LIN {X 0,Y 361.818,Z 305.412,A -85,B 0,C 180,E1 -12994.284,E2 -12994.284} C_VEL
LIN {X 0,Y 361.885,Z 305.409,A -85,B 0,C 180,E1 -12997.238,E2 -12997.238} C_VEL
LIN {X 0,Y 361.874,Z 305.407,A -85,B 0,C 180,E1 -13000.773,E2 -13000.773} C_VEL
LIN {X 0,Y 361.905,Z 305.409,A -85,B 0,C 180,E1 -13004.355,E2 -13004.355} C_VEL
LIN {X 0,Y 361.86,Z 305.417,A -85,B 0,C 180,E1 -13007.564,E2 -13007.564} C_VEL
LIN {X 0,Y 361.852,Z 305.412,A -85,B 0,C 180,E1 -13010.977,E2 -13010.977} C_VEL
LIN {X 0,Y 361.854,Z 305.412,A -85,B 0,C 180,E1 -13014.66,E2 -13014.66} C_VEL
LIN {X 0,Y 361.82,Z 305.42,A -85,B 0,C 180,E1 -13018.376,E2 -13018.376} C_VEL
LIN {X 0,Y 361.917,Z 305.621,A -85,B 0,C 180,E1 -13019.606,E2 -13019.606} C_VEL
LIN {X 0,Y 364.515,Z 316.864,A -85,B 0,C 180,E1 -13022.487,E2 -13022.487} C_VEL
LIN {X 0,Y 366.087,Z 325.864,A -85,B 0,C 180,E1 -13024.673,E2 -13024.673} C_VEL
LIN {X 0,Y 364.917,Z 338.677,A -85,B 0,C 180,E1 -13027.483,E2 -13027.483} C_VEL
LIN {X 0,Y 368.842,Z 360.352,A -85,B 0,C 180,E1 -13028.244,E2 -13028.244} C_VEL
LIN {X 0,Y 370.844,Z 375.541,A -85,B 0,C 180,E1 -13028.711,E2 -13028.711} C_VEL
LIN {X 0,Y 369.356,Z 448.545,A -85,B 0,C 180,E1 -13030.23,E2 -13030.23} C_VEL
LIN {X 0,Y 368.568,Z 462.077,A -85,B 0,C 180,E1 -13030.729,E2 -13030.729} C_VEL
LIN {X 0,Y 367.613,Z 474.38,A -85,B 0,C 180,E1 -13031.401,E2 -13031.401} C_VEL
LIN {X 0,Y 366.546,Z 486.228,A -85,B 0,C 180,E1 -13032.284,E2 -13032.284} C_VEL
LIN {X 0,Y 365.417,Z 497.657,A -85,B 0,C 180,E1 -13033.381,E2 -13033.381} C_VEL
LIN {X 0,Y 364.385,Z 507.488,A -85,B 0,C 180,E1 -13034.557,E2 -13034.557} C_VEL
LIN {X 0,Y 363.289,Z 517.316,A -85,B 0,C 180,E1 -13036.011,E2 -13036.011} C_VEL
LIN {X 0,Y 362.23,Z 526.378,A -85,B 0,C 180,E1 -13037.682,E2 -13037.682} C_VEL
LIN {X 0,Y 361.454,Z 533.695,A -85,B 0,C 180,E1 -13039.36,E2 -13039.36} C_VEL
LIN {X 0,Y 360.909,Z 539.555,A -85,B 0,C 180,E1 -13041.042,E2 -13041.042} C_VEL
LIN {X 0,Y 360.588,Z 544.181,A -85,B 0,C 180,E1 -13042.726,E2 -13042.726} C_VEL
LIN {X 0,Y 360.381,Z 547.708,A -85,B 0,C 180,E1 -13044.408,E2 -13044.408} C_VEL
LIN {X 0,Y 360.364,Z 549.477,A -85,B 0,C 180,E1 -13045.53,E2 -13045.53} C_VEL
LIN {X 0,Y 360.298,Z 551.789,A -85,B 0,C 180,E1 -13047.768,E2 -13047.768} C_VEL
LIN {X 0,Y 360.369,Z 552.341,A -85,B 0,C 180,E1 -13048.886,E2 -13048.886} C_VEL
LIN {X 0,Y 360.424,Z 552.454,A -85,B 0,C 180,E1 -13050.004,E2 -13050.004} C_VEL
LIN {X 0,Y 360.386,Z 552.17,A -85,B 0,C 180,E1 -13051.121,E2 -13051.121} C_VEL
LIN {X 0,Y 360.303,Z 551.492,A -85,B 0,C 180,E1 -13052.239,E2 -13052.239} C_VEL
LIN {X 0,Y 360.305,Z 550.405,A -85,B 0,C 180,E1 -13053.358,E2 -13053.358} C_VEL
LIN {X 0,Y 360.367,Z 548.86,A -85,B 0,C 180,E1 -13054.477,E2 -13054.477} C_VEL
LIN {X 0,Y 360.38,Z 546.171,A -85,B 0,C 180,E1 -13055.964,E2 -13055.964} C_VEL
LIN {X 0,Y 360.652,Z 541.532,A -85,B 0,C 180,E1 -13057.843,E2 -13057.843} C_VEL
LIN {X 0,Y 361.083,Z 535.11,A -85,B 0,C 180,E1 -13059.809,E2 -13059.809} C_VEL
LIN {X 0,Y 361.669,Z 528.101,A -85,B 0,C 180,E1 -13061.492,E2 -13061.492} C_VEL
LIN {X 0,Y 362.597,Z 519.308,A -85,B 0,C 180,E1 -13063.167,E2 -13063.167} C_VEL
LIN {X 0,Y 363.604,Z 509.036,A -85,B 0,C 180,E1 -13064.738,E2 -13064.738} C_VEL
LIN {X 0,Y 364.589,Z 497.831,A -85,B 0,C 180,E1 -13066.09,E2 -13066.09} C_VEL
LIN {X 0,Y 365.697,Z 486.255,A -85,B 0,C 180,E1 -13067.189,E2 -13067.189} C_VEL
LIN {X 0,Y 366.655,Z 474.067,A -85,B 0,C 180,E1 -13068.079,E2 -13068.079} C_VEL
LIN {X 0,Y 367.595,Z 460.562,A -85,B 0,C 180,E1 -13068.788,E2 -13068.788} C_VEL
LIN {X 0,Y 368.122,Z 448.077,A -85,B 0,C 180,E1 -13069.23,E2 -13069.23} C_VEL
LIN {X 0,Y 369.425,Z 373.616,A -85,B 0,C 180,E1 -13070.75,E2 -13070.75} C_VEL
LIN {X 0,Y 364.371,Z 340.015,A -85,B 0,C 180,E1 -13071.754,E2 -13071.754} C_VEL
LIN {X 0,Y 365.678,Z 325.548,A -85,B 0,C 180,E1 -13075.015,E2 -13075.015} C_VEL
LIN {X 0,Y 365.209,Z 321.353,A -85,B 0,C 180,E1 -13076.022,E2 -13076.022} C_VEL
LIN {X 0,Y 363.128,Z 310.962,A -85,B 0,C 180,E1 -13078.623,E2 -13078.623} C_VEL
LIN {X 0,Y 361.897,Z 305.409,A -85,B 0,C 180,E1 -13080.106,E2 -13080.106} C_VEL
LIN {X 0,Y 361.86,Z 305.412,A -85,B 0,C 180,E1 -13084.281,E2 -13084.281} C_VEL
LIN {X 0,Y 361.867,Z 305.405,A -85,B 0,C 180,E1 -13087.223,E2 -13087.223} C_VEL
LIN {X 0,Y 361.839,Z 305.411,A -85,B 0,C 180,E1 -13090.756,E2 -13090.756} C_VEL
LIN {X 0,Y 361.82,Z 305.418,A -85,B 0,C 180,E1 -13094.369,E2 -13094.369} C_VEL
LIN {X 0,Y 361.839,Z 305.409,A -85,B 0,C 180,E1 -13097.569,E2 -13097.569} C_VEL
LIN {X 0,Y 361.871,Z 305.407,A -85,B 0,C 180,E1 -13100.974,E2 -13100.974} C_VEL
LIN {X 0,Y 361.875,Z 305.411,A -85,B 0,C 180,E1 -13104.656,E2 -13104.656} C_VEL
LIN {X 0,Y 361.838,Z 305.412,A -85,B 0,C 180,E1 -13108.371,E2 -13108.371} C_VEL
LIN {X 0,Y 361.908,Z 305.401,A -85,B 0,C 180,E1 -13112.221,E2 -13112.221} C_VEL
LIN {X 0,Y 361.927,Z 305.403,A -85,B 0,C 180,E1 -13114.71,E2 -13114.71} C_VEL
LIN {X 0,Y 361.861,Z 305.407,A -85,B 0,C 180,E1 -13118.345,E2 -13118.345} C_VEL
LIN {X 0,Y 361.919,Z 305.399,A -85,B 0,C 180,E1 -13122.085,E2 -13122.085} C_VEL
LIN {X 0,Y 361.959,Z 305.398,A -85,B 0,C 180,E1 -13125.379,E2 -13125.379} C_VEL
LIN {X 0,Y 361.966,Z 305.395,A -85,B 0,C 180,E1 -13128.804,E2 -13128.804} C_VEL
LIN {X 0,Y 362.114,Z 305.374,A -85,B 0,C 180,E1 -13132.192,E2 -13132.192} C_VEL
LIN {X 0,Y 362.108,Z 305.375,A -85,B 0,C 180,E1 -13134.431,E2 -13134.431} C_VEL
LIN {X 0,Y 362.273,Z 305.358,A -85,B 0,C 180,E1 -13137.776,E2 -13137.776} C_VEL
LIN {X 0,Y 362.377,Z 305.343,A -85,B 0,C 180,E1 -13140,E2 -13140} C_VEL
LIN {X 0,Y 362.273,Z 305.355,A -85,B 0,C 180,E1 -13142.224,E2 -13142.224} C_VEL
LIN {X 0,Y 362.119,Z 305.374,A -85,B 0,C 180,E1 -13146.687,E2 -13146.687} C_VEL
LIN {X 0,Y 361.995,Z 305.392,A -85,B 0,C 180,E1 -13150.063,E2 -13150.063} C_VEL
LIN {X 0,Y 361.996,Z 305.395,A -85,B 0,C 180,E1 -13153.898,E2 -13153.898} C_VEL
LIN {X 0,Y 361.925,Z 305.398,A -85,B 0,C 180,E1 -13156.934,E2 -13156.934} C_VEL
LIN {X 0,Y 361.882,Z 305.405,A -85,B 0,C 180,E1 -13160.461,E2 -13160.461} C_VEL
LIN {X 0,Y 361.861,Z 305.413,A -85,B 0,C 180,E1 -13164.101,E2 -13164.101} C_VEL
LIN {X 0,Y 361.834,Z 305.412,A -85,B 0,C 180,E1 -13167.785,E2 -13167.785} C_VEL
LIN {X 0,Y 361.827,Z 305.41,A -85,B 0,C 180,E1 -13171.279,E2 -13171.279} C_VEL
LIN {X 0,Y 361.851,Z 305.414,A -85,B 0,C 180,E1 -13174.281,E2 -13174.281} C_VEL
LIN {X 0,Y 361.856,Z 305.407,A -85,B 0,C 180,E1 -13177.221,E2 -13177.221} C_VEL
LIN {X 0,Y 361.811,Z 305.416,A -85,B 0,C 180,E1 -13180.75,E2 -13180.75} C_VEL
LIN {X 0,Y 361.801,Z 305.418,A -85,B 0,C 180,E1 -13184.371,E2 -13184.371} C_VEL
LIN {X 0,Y 361.814,Z 305.412,A -85,B 0,C 180,E1 -13187.572,E2 -13187.572} C_VEL
LIN {X 0,Y 361.824,Z 305.414,A -85,B 0,C 180,E1 -13190.983,E2 -13190.983} C_VEL
LIN {X 0,Y 361.841,Z 305.414,A -85,B 0,C 180,E1 -13194.663,E2 -13194.663} C_VEL
LIN {X 0,Y 361.816,Z 305.413,A -85,B 0,C 180,E1 -13198.367,E2 -13198.367} C_VEL
LIN {X 0,Y 361.855,Z 305.414,A -85,B 0,C 180,E1 -13200.949,E2 -13200.949} C_VEL
LIN {X 0,Y 361.884,Z 305.406,A -85,B 0,C 180,E1 -13204.705,E2 -13204.705} C_VEL
LIN {X 0,Y 361.86,Z 305.406,A -85,B 0,C 180,E1 -13208.343,E2 -13208.343} C_VEL
LIN {X 0,Y 361.927,Z 305.398,A -85,B 0,C 180,E1 -13212.083,E2 -13212.083} C_VEL
LIN {X 0,Y 361.967,Z 305.399,A -85,B 0,C 180,E1 -13215.377,E2 -13215.377} C_VEL
LIN {X 0,Y 361.973,Z 305.393,A -85,B 0,C 180,E1 -13218.802,E2 -13218.802} C_VEL
LIN {X 0,Y 362.082,Z 305.379,A -85,B 0,C 180,E1 -13222.188,E2 -13222.188} C_VEL
LIN {X 0,Y 362.092,Z 305.377,A -85,B 0,C 180,E1 -13224.428,E2 -13224.428} C_VEL
LIN {X 0,Y 362.266,Z 305.36,A -85,B 0,C 180,E1 -13227.773,E2 -13227.773} C_VEL
LIN {X 0,Y 362.176,Z 305.368,A -85,B 0,C 180,E1 -13231.108,E2 -13231.108} C_VEL
LIN {X 0,Y 362.267,Z 305.357,A -85,B 0,C 180,E1 -13232.22,E2 -13232.22} C_VEL
LIN {X 0,Y 362.114,Z 305.379,A -85,B 0,C 180,E1 -13236.683,E2 -13236.683} C_VEL
LIN {X 0,Y 362.084,Z 305.457,A -85,B 0,C 180,E1 -13237.735,E2 -13237.735} C_VEL
LIN {X 0,Y 363.779,Z 314.594,A -85,B 0,C 180,E1 -13240.271,E2 -13240.271} C_VEL
LIN {X 0,Y 366.864,Z 324.402,A -85,B 0,C 180,E1 -13240.675,E2 -13240.675} C_VEL
LIN {X 0,Y 369.922,Z 340.115,A -85,B 0,C 180,E1 -13241.181,E2 -13241.181} C_VEL
LIN {X 0,Y 368.349,Z 422.054,A -85,B 0,C 180,E1 -13242.85,E2 -13242.85} C_VEL
LIN {X 0,Y 367.824,Z 435.697,A -85,B 0,C 180,E1 -13243.356,E2 -13243.356} C_VEL
LIN {X 0,Y 367.154,Z 448.332,A -85,B 0,C 180,E1 -13244.051,E2 -13244.051} C_VEL
LIN {X 0,Y 366.4,Z 459.282,A -85,B 0,C 180,E1 -13244.861,E2 -13244.861} C_VEL
LIN {X 0,Y 365.344,Z 471.437,A -85,B 0,C 180,E1 -13246.019,E2 -13246.019} C_VEL
LIN {X 0,Y 364.346,Z 481.673,A -85,B 0,C 180,E1 -13247.247,E2 -13247.247} C_VEL
LIN {X 0,Y 363.485,Z 491.125,A -85,B 0,C 180,E1 -13248.662,E2 -13248.662} C_VEL
LIN {X 0,Y 362.672,Z 499.049,A -85,B 0,C 180,E1 -13250.113,E2 -13250.113} C_VEL
LIN {X 0,Y 361.84,Z 507.132,A -85,B 0,C 180,E1 -13251.95,E2 -13251.95} C_VEL
LIN {X 0,Y 361.399,Z 512.236,A -85,B 0,C 180,E1 -13253.409,E2 -13253.409} C_VEL
LIN {X 0,Y 360.46,Z 514.812,A -85,B 0,C 180,E1 -13254.246,E2 -13254.246} C_VEL
LIN {X 0,Y 357.241,Z 518.482,A -85,B 0,C 180,E1 -13255.627,E2 -13255.627} C_VEL
LIN {X 0,Y 354.605,Z 520.942,A -85,B 0,C 180,E1 -13256.772,E2 -13256.772} C_VEL
LIN {X 0,Y 353.342,Z 522.719,A -85,B 0,C 180,E1 -13257.835,E2 -13257.835} C_VEL
LIN {X 0,Y 353.298,Z 522.853,A -85,B 0,C 180,E1 -13257.99,E2 -13257.99} C_VEL
LIN {X 0,Y 353.135,Z 524.909,A -85,B 0,C 180,E1 -13259.831,E2 -13259.831} C_VEL
LIN {X 0,Y 353.076,Z 525.685,A -85,B 0,C 180,E1 -13261.16,E2 -13261.16} C_VEL
LIN {X 0,Y 353.079,Z 525.823,A -85,B 0,C 180,E1 -13263.279,E2 -13263.279} C_VEL
LIN {X 0,Y 353.265,Z 524.589,A -85,B 0,C 180,E1 -13265.346,E2 -13265.346} C_VEL
LIN {X 0,Y 353.584,Z 522.143,A -85,B 0,C 180,E1 -13267.339,E2 -13267.339} C_VEL
LIN {X 0,Y 354.059,Z 518.189,A -85,B 0,C 180,E1 -13269.426,E2 -13269.426} C_VEL
LIN {X 0,Y 354.54,Z 513.776,A -85,B 0,C 180,E1 -13271.125,E2 -13271.125} C_VEL
LIN {X 0,Y 355.306,Z 507.655,A -85,B 0,C 180,E1 -13272.957,E2 -13272.957} C_VEL
LIN {X 0,Y 356.28,Z 500.017,A -85,B 0,C 180,E1 -13274.754,E2 -13274.754} C_VEL
LIN {X 0,Y 357.319,Z 492.288,A -85,B 0,C 180,E1 -13276.22,E2 -13276.22} C_VEL
LIN {X 0,Y 358.533,Z 482.581,A -85,B 0,C 180,E1 -13277.72,E2 -13277.72} C_VEL
LIN {X 0,Y 359.62,Z 471.967,A -85,B 0,C 180,E1 -13279.03,E2 -13279.03} C_VEL
LIN {X 0,Y 360.855,Z 460.512,A -85,B 0,C 180,E1 -13280.145,E2 -13280.145} C_VEL
LIN {X 0,Y 361.828,Z 448.47,A -85,B 0,C 180,E1 -13281.052,E2 -13281.052} C_VEL
LIN {X 0,Y 362.581,Z 435.556,A -85,B 0,C 180,E1 -13281.765,E2 -13281.765} C_VEL
LIN {X 0,Y 363.169,Z 422.591,A -85,B 0,C 180,E1 -13282.243,E2 -13282.243} C_VEL
LIN {X 0,Y 364.894,Z 340.765,A -85,B 0,C 180,E1 -13283.969,E2 -13283.969} C_VEL
LIN {X 0,Y 362.053,Z 327.901,A -85,B 0,C 180,E1 -13284.47,E2 -13284.47} C_VEL
LIN {X 0,Y 356.857,Z 315.027,A -85,B 0,C 180,E1 -13285.171,E2 -13285.171} C_VEL
LIN {X 0,Y 354.77,Z 306.294,A -85,B 0,C 180,E1 -13287.539,E2 -13287.539} C_VEL
LIN {X 0,Y 354.831,Z 306.29,A -85,B 0,C 180,E1 -13290.618,E2 -13290.618} C_VEL
LIN {X 0,Y 354.858,Z 306.29,A -85,B 0,C 180,E1 -13294.169,E2 -13294.169} C_VEL
LIN {X 0,Y 354.786,Z 306.298,A -85,B 0,C 180,E1 -13297.891,E2 -13297.891} C_VEL
LIN {X 0,Y 354.879,Z 306.28,A -85,B 0,C 180,E1 -13301.89,E2 -13301.89} C_VEL
LIN {X 0,Y 354.897,Z 306.277,A -85,B 0,C 180,E1 -13305.98,E2 -13305.98} C_VEL
LIN {X 0,Y 354.91,Z 306.27,A -85,B 0,C 180,E1 -13309.734,E2 -13309.734} C_VEL
LIN {X 0,Y 355.077,Z 306.253,A -85,B 0,C 180,E1 -13313.18,E2 -13313.18} C_VEL
LIN {X 0,Y 355.198,Z 306.237,A -85,B 0,C 180,E1 -13317.732,E2 -13317.732} C_VEL
LIN {X 0,Y 355.328,Z 306.214,A -85,B 0,C 180,E1 -13320,E2 -13320} C_VEL
LIN {X 0,Y 355.199,Z 306.238,A -85,B 0,C 180,E1 -13322.268,E2 -13322.268} C_VEL
LIN {X 0,Y 355.08,Z 306.252,A -85,B 0,C 180,E1 -13326.82,E2 -13326.82} C_VEL
LIN {X 0,Y 354.936,Z 306.271,A -85,B 0,C 180,E1 -13330.265,E2 -13330.265} C_VEL
LIN {X 0,Y 354.897,Z 306.275,A -85,B 0,C 180,E1 -13334.02,E2 -13334.02} C_VEL
LIN {X 0,Y 354.88,Z 306.275,A -85,B 0,C 180,E1 -13338.111,E2 -13338.111} C_VEL
LIN {X 0,Y 354.818,Z 306.282,A -85,B 0,C 180,E1 -13342.107,E2 -13342.107} C_VEL
LIN {X 0,Y 354.859,Z 306.28,A -85,B 0,C 180,E1 -13345.831,E2 -13345.831} C_VEL
LIN {X 0,Y 354.816,Z 306.288,A -85,B 0,C 180,E1 -13349.682,E2 -13349.682} C_VEL
LIN {X 0,Y 354.771,Z 306.294,A -85,B 0,C 180,E1 -13353.706,E2 -13353.706} C_VEL
LIN {X 0,Y 354.844,Z 306.283,A -85,B 0,C 180,E1 -13357.616,E2 -13357.616} C_VEL
LIN {X 0,Y 354.825,Z 306.286,A -85,B 0,C 180,E1 -13360.816,E2 -13360.816} C_VEL
LIN {X 0,Y 354.859,Z 306.286,A -85,B 0,C 180,E1 -13364.531,E2 -13364.531} C_VEL
LIN {X 0,Y 354.814,Z 306.293,A -85,B 0,C 180,E1 -13367.674,E2 -13367.674} C_VEL
LIN {X 0,Y 354.814,Z 306.289,A -85,B 0,C 180,E1 -13370.674,E2 -13370.674} C_VEL
LIN {X 0,Y 354.801,Z 306.287,A -85,B 0,C 180,E1 -13374.306,E2 -13374.306} C_VEL
LIN {X 0,Y 354.769,Z 306.303,A -85,B 0,C 180,E1 -13377.672,E2 -13377.672} C_VEL
LIN {X 0,Y 354.861,Z 306.472,A -85,B 0,C 180,E1 -13379.15,E2 -13379.15} C_VEL
LIN {X 0,Y 357.554,Z 318.013,A -85,B 0,C 180,E1 -13382.192,E2 -13382.192} C_VEL
LIN {X 0,Y 359.229,Z 327.337,A -85,B 0,C 180,E1 -13384.512,E2 -13384.512} C_VEL
LIN {X 0,Y 358.128,Z 338.37,A -85,B 0,C 180,E1 -13386.974,E2 -13386.974} C_VEL
LIN {X 0,Y 362.315,Z 360.994,A -85,B 0,C 180,E1 -13387.808,E2 -13387.808} C_VEL
LIN {X 0,Y 364.338,Z 375.808,A -85,B 0,C 180,E1 -13388.28,E2 -13388.28} C_VEL
LIN {X 0,Y 362.759,Z 448.376,A -85,B 0,C 180,E1 -13389.818,E2 -13389.818} C_VEL
LIN {X 0,Y 361.959,Z 461.864,A -85,B 0,C 180,E1 -13390.326,E2 -13390.326} C_VEL
LIN {X 0,Y 360.906,Z 474.652,A -85,B 0,C 180,E1 -13391.042,E2 -13391.042} C_VEL
LIN {X 0,Y 359.816,Z 486.378,A -85,B 0,C 180,E1 -13391.941,E2 -13391.941} C_VEL
LIN {X 0,Y 358.623,Z 497.725,A -85,B 0,C 180,E1 -13393.057,E2 -13393.057} C_VEL
LIN {X 0,Y 357.488,Z 507.837,A -85,B 0,C 180,E1 -13394.3,E2 -13394.3} C_VEL
LIN {X 0,Y 356.363,Z 517.236,A -85,B 0,C 180,E1 -13395.733,E2 -13395.733} C_VEL
LIN {X 0,Y 355.271,Z 526.256,A -85,B 0,C 180,E1 -13397.436,E2 -13397.436} C_VEL
LIN {X 0,Y 354.419,Z 533.544,A -85,B 0,C 180,E1 -13399.146,E2 -13399.146} C_VEL
LIN {X 0,Y 353.865,Z 539.378,A -85,B 0,C 180,E1 -13400.862,E2 -13400.862} C_VEL
LIN {X 0,Y 353.51,Z 543.983,A -85,B 0,C 180,E1 -13402.58,E2 -13402.58} C_VEL
LIN {X 0,Y 353.287,Z 547.494,A -85,B 0,C 180,E1 -13404.296,E2 -13404.296} C_VEL
LIN {X 0,Y 353.277,Z 549.251,A -85,B 0,C 180,E1 -13405.44,E2 -13405.44} C_VEL
LIN {X 0,Y 353.223,Z 550.597,A -85,B 0,C 180,E1 -13406.582,E2 -13406.582} C_VEL
LIN {X 0,Y 353.203,Z 551.546,A -85,B 0,C 180,E1 -13407.723,E2 -13407.723} C_VEL
LIN {X 0,Y 353.269,Z 552.081,A -85,B 0,C 180,E1 -13408.864,E2 -13408.864} C_VEL
LIN {X 0,Y 353.329,Z 552.183,A -85,B 0,C 180,E1 -13410.004,E2 -13410.004} C_VEL
LIN {X 0,Y 353.286,Z 551.89,A -85,B 0,C 180,E1 -13411.143,E2 -13411.143} C_VEL
LIN {X 0,Y 353.208,Z 551.202,A -85,B 0,C 180,E1 -13412.284,E2 -13412.284} C_VEL
LIN {X 0,Y 353.226,Z 550.096,A -85,B 0,C 180,E1 -13413.425,E2 -13413.425} C_VEL
LIN {X 0,Y 353.279,Z 548.538,A -85,B 0,C 180,E1 -13414.568,E2 -13414.568} C_VEL
LIN {X 0,Y 353.298,Z 546.122,A -85,B 0,C 180,E1 -13415.94,E2 -13415.94} C_VEL
LIN {X 0,Y 353.509,Z 542.696,A -85,B 0,C 180,E1 -13417.428,E2 -13417.428} C_VEL
LIN {X 0,Y 353.825,Z 537.689,A -85,B 0,C 180,E1 -13419.146,E2 -13419.146} C_VEL
LIN {X 0,Y 354.334,Z 531.382,A -85,B 0,C 180,E1 -13420.864,E2 -13420.864} C_VEL
LIN {X 0,Y 355.152,Z 523.483,A -85,B 0,C 180,E1 -13422.575,E2 -13422.575} C_VEL
LIN {X 0,Y 355.985,Z 515.412,A -85,B 0,C 180,E1 -13423.998,E2 -13423.998} C_VEL
LIN {X 0,Y 356.98,Z 505.448,A -85,B 0,C 180,E1 -13425.431,E2 -13425.431} C_VEL
LIN {X 0,Y 358.019,Z 494.582,A -85,B 0,C 180,E1 -13426.687,E2 -13426.687} C_VEL
LIN {X 0,Y 359.162,Z 482.061,A -85,B 0,C 180,E1 -13427.806,E2 -13427.806} C_VEL
LIN {X 0,Y 360.153,Z 469.789,A -85,B 0,C 180,E1 -13428.638,E2 -13428.638} C_VEL
LIN {X 0,Y 360.946,Z 456.887,A -85,B 0,C 180,E1 -13429.259,E2 -13429.259} C_VEL
LIN {X 0,Y 361.503,Z 443.35,A -85,B 0,C 180,E1 -13429.671,E2 -13429.671} C_VEL
LIN {X 0,Y 362.658,Z 374.276,A -85,B 0,C 180,E1 -13431.097,E2 -13431.097} C_VEL
LIN {X 0,Y 357.485,Z 339.682,A -85,B 0,C 180,E1 -13432.174,E2 -13432.174} C_VEL
LIN {X 0,Y 358.732,Z 326.411,A -85,B 0,C 180,E1 -13435.223,E2 -13435.223} C_VEL
LIN {X 0,Y 357.763,Z 319.8,A -85,B 0,C 180,E1 -13436.862,E2 -13436.862} C_VEL
LIN {X 0,Y 354.862,Z 306.286,A -85,B 0,C 180,E1 -13440.417,E2 -13440.417} C_VEL
LIN {X 0,Y 354.812,Z 306.286,A -85,B 0,C 180,E1 -13443.703,E2 -13443.703} C_VEL
LIN {X 0,Y 354.803,Z 306.289,A -85,B 0,C 180,E1 -13446.461,E2 -13446.461} C_VEL
LIN {X 0,Y 354.83,Z 306.282,A -85,B 0,C 180,E1 -13449.424,E2 -13449.424} C_VEL
LIN {X 0,Y 354.792,Z 306.288,A -85,B 0,C 180,E1 -13452.868,E2 -13452.868} C_VEL
LIN {X 0,Y 354.77,Z 306.292,A -85,B 0,C 180,E1 -13456.104,E2 -13456.104} C_VEL
LIN {X 0,Y 354.79,Z 306.288,A -85,B 0,C 180,E1 -13459.179,E2 -13459.179} C_VEL
LIN {X 0,Y 354.809,Z 306.289,A -85,B 0,C 180,E1 -13462.403,E2 -13462.403} C_VEL
LIN {X 0,Y 354.813,Z 306.288,A -85,B 0,C 180,E1 -13464.941,E2 -13464.941} C_VEL
LIN {X 0,Y 354.794,Z 306.289,A -85,B 0,C 180,E1 -13468.406,E2 -13468.406} C_VEL
LIN {X 0,Y 354.847,Z 306.28,A -85,B 0,C 180,E1 -13471.619,E2 -13471.619} C_VEL
LIN {X 0,Y 354.898,Z 306.274,A -85,B 0,C 180,E1 -13474.172,E2 -13474.172} C_VEL
LIN {X 0,Y 354.816,Z 306.284,A -85,B 0,C 180,E1 -13477.893,E2 -13477.893} C_VEL
LIN {X 0,Y 354.889,Z 306.275,A -85,B 0,C 180,E1 -13481.908,E2 -13481.908} C_VEL
LIN {X 0,Y 354.941,Z 306.268,A -85,B 0,C 180,E1 -13485.982,E2 -13485.982} C_VEL
LIN {X 0,Y 354.954,Z 306.268,A -85,B 0,C 180,E1 -13489.735,E2 -13489.735} C_VEL
LIN {X 0,Y 355.121,Z 306.251,A -85,B 0,C 180,E1 -13493.18,E2 -13493.18} C_VEL
LIN {X 0,Y 355.237,Z 306.235,A -85,B 0,C 180,E1 -13497.732,E2 -13497.732} C_VEL
LIN {X 0,Y 355.328,Z 306.221,A -85,B 0,C 180,E1 -13500,E2 -13500} C_VEL
LIN {X 0,Y 355.237,Z 306.232,A -85,B 0,C 180,E1 -13502.268,E2 -13502.268} C_VEL
LIN {X 0,Y 355.084,Z 306.25,A -85,B 0,C 180,E1 -13506.82,E2 -13506.82} C_VEL
LIN {X 0,Y 354.952,Z 306.268,A -85,B 0,C 180,E1 -13510.265,E2 -13510.265} C_VEL
LIN {X 0,Y 354.941,Z 306.273,A -85,B 0,C 180,E1 -13514.018,E2 -13514.018} C_VEL
LIN {X 0,Y 354.889,Z 306.279,A -85,B 0,C 180,E1 -13518.092,E2 -13518.092} C_VEL
LIN {X 0,Y 354.804,Z 306.291,A -85,B 0,C 180,E1 -13522.108,E2 -13522.108} C_VEL
LIN {X 0,Y 354.794,Z 306.29,A -85,B 0,C 180,E1 -13525.836,E2 -13525.836} C_VEL
LIN {X 0,Y 354.786,Z 306.289,A -85,B 0,C 180,E1 -13529.685,E2 -13529.685} C_VEL
LIN {X 0,Y 354.809,Z 306.286,A -85,B 0,C 180,E1 -13533.702,E2 -13533.702} C_VEL
LIN {X 0,Y 354.792,Z 306.292,A -85,B 0,C 180,E1 -13536.46,E2 -13536.46} C_VEL
LIN {X 0,Y 354.771,Z 306.289,A -85,B 0,C 180,E1 -13539.412,E2 -13539.412} C_VEL
LIN {X 0,Y 354.78,Z 306.291,A -85,B 0,C 180,E1 -13542.865,E2 -13542.865} C_VEL
LIN {X 0,Y 354.741,Z 306.295,A -85,B 0,C 180,E1 -13546.098,E2 -13546.098} C_VEL
LIN {X 0,Y 354.765,Z 306.292,A -85,B 0,C 180,E1 -13549.174,E2 -13549.174} C_VEL
LIN {X 0,Y 354.787,Z 306.29,A -85,B 0,C 180,E1 -13552.407,E2 -13552.407} C_VEL
LIN {X 0,Y 354.776,Z 306.294,A -85,B 0,C 180,E1 -13554.935,E2 -13554.935} C_VEL
LIN {X 0,Y 354.772,Z 306.291,A -85,B 0,C 180,E1 -13558.411,E2 -13558.411} C_VEL
LIN {X 0,Y 354.794,Z 306.287,A -85,B 0,C 180,E1 -13561.612,E2 -13561.612} C_VEL
LIN {X 0,Y 354.84,Z 306.282,A -85,B 0,C 180,E1 -13565.656,E2 -13565.656} C_VEL
LIN {X 0,Y 354.833,Z 306.288,A -85,B 0,C 180,E1 -13569.111,E2 -13569.111} C_VEL
LIN {X 0,Y 354.886,Z 306.277,A -85,B 0,C 180,E1 -13572.717,E2 -13572.717} C_VEL
LIN {X 0,Y 354.957,Z 306.266,A -85,B 0,C 180,E1 -13576.253,E2 -13576.253} C_VEL
LIN {X 0,Y 354.958,Z 306.269,A -85,B 0,C 180,E1 -13579.732,E2 -13579.732} C_VEL
LIN {X 0,Y 355.089,Z 306.253,A -85,B 0,C 180,E1 -13583.177,E2 -13583.177} C_VEL
LIN {X 0,Y 355.229,Z 306.237,A -85,B 0,C 180,E1 -13587.729,E2 -13587.729} C_VEL
LIN {X 0,Y 355.147,Z 306.244,A -85,B 0,C 180,E1 -13591.13,E2 -13591.13} C_VEL
LIN {X 0,Y 355.229,Z 306.233,A -85,B 0,C 180,E1 -13592.264,E2 -13592.264} C_VEL
LIN {X 0,Y 355.079,Z 306.255,A -85,B 0,C 180,E1 -13596.816,E2 -13596.816} C_VEL
LIN {X 0,Y 355.038,Z 306.425,A -85,B 0,C 180,E1 -13597.46,E2 -13597.46} C_VEL
LIN {X 0,Y 356.696,Z 315.172,A -85,B 0,C 180,E1 -13599.884,E2 -13599.884} C_VEL
LIN {X 0,Y 360.429,Z 326.619,A -85,B 0,C 180,E1 -13600.355,E2 -13600.355} C_VEL
LIN {X 0,Y 363.224,Z 341.58,A -85,B 0,C 180,E1 -13600.841,E2 -13600.841} C_VEL
LIN {X 0,Y 361.555,Z 422.92,A -85,B 0,C 180,E1 -13602.535,E2 -13602.535} C_VEL
LIN {X 0,Y 361.012,Z 436.623,A -85,B 0,C 180,E1 -13603.063,E2 -13603.063} C_VEL
LIN {X 0,Y 360.333,Z 448.699,A -85,B 0,C 180,E1 -13603.747,E2 -13603.747} C_VEL
LIN {X 0,Y 359.556,Z 459.617,A -85,B 0,C 180,E1 -13604.571,E2 -13604.571} C_VEL
LIN {X 0,Y 358.556,Z 470.653,A -85,B 0,C 180,E1 -13605.63,E2 -13605.63} C_VEL
LIN {X 0,Y 357.465,Z 481.855,A -85,B 0,C 180,E1 -13606.985,E2 -13606.985} C_VEL
LIN {X 0,Y 356.6,Z 491.031,A -85,B 0,C 180,E1 -13608.376,E2 -13608.376} C_VEL
LIN {X 0,Y 355.685,Z 499.347,A -85,B 0,C 180,E1 -13609.923,E2 -13609.923} C_VEL
LIN {X 0,Y 354.839,Z 507.208,A -85,B 0,C 180,E1 -13611.74,E2 -13611.74} C_VEL
LIN {X 0,Y 354.344,Z 512.793,A -85,B 0,C 180,E1 -13613.365,E2 -13613.365} C_VEL
LIN {X 0,Y 353.843,Z 517.933,A -85,B 0,C 180,E1 -13615.273,E2 -13615.273} C_VEL
LIN {X 0,Y 353.442,Z 521.739,A -85,B 0,C 180,E1 -13617.21,E2 -13617.21} C_VEL
LIN {X 0,Y 353.298,Z 522.853,A -85,B 0,C 180,E1 -13617.99,E2 -13617.99} C_VEL
LIN {X 0,Y 352.513,Z 524.096,A -85,B 0,C 180,E1 -13618.92,E2 -13618.92} C_VEL
LIN {X 0,Y 349.512,Z 525.486,A -85,B 0,C 180,E1 -13620.446,E2 -13620.446} C_VEL
LIN {X 0,Y 347.056,Z 526.065,A -85,B 0,C 180,E1 -13621.692,E2 -13621.692} C_VEL
LIN {X 0,Y 346.046,Z 526.177,A -85,B 0,C 180,E1 -13622.66,E2 -13622.66} C_VEL
LIN {X 0,Y 345.985,Z 526.114,A -85,B 0,C 180,E1 -13622.988,E2 -13622.988} C_VEL
LIN {X 0,Y 346.093,Z 525.472,A -85,B 0,C 180,E1 -13624.644,E2 -13624.644} C_VEL
LIN {X 0,Y 346.278,Z 524.291,A -85,B 0,C 180,E1 -13626.049,E2 -13626.049} C_VEL
LIN {X 0,Y 346.673,Z 521.119,A -85,B 0,C 180,E1 -13628.276,E2 -13628.276} C_VEL
LIN {X 0,Y 347.242,Z 516.699,A -85,B 0,C 180,E1 -13630.357,E2 -13630.357} C_VEL
LIN {X 0,Y 347.898,Z 511.49,A -85,B 0,C 180,E1 -13632.189,E2 -13632.189} C_VEL
LIN {X 0,Y 348.822,Z 504.634,A -85,B 0,C 180,E1 -13634.06,E2 -13634.06} C_VEL
LIN {X 0,Y 349.875,Z 497.053,A -85,B 0,C 180,E1 -13635.71,E2 -13635.71} C_VEL
LIN {X 0,Y 351.132,Z 487.729,A -85,B 0,C 180,E1 -13637.347,E2 -13637.347} C_VEL
LIN {X 0,Y 352.296,Z 477.92,A -85,B 0,C 180,E1 -13638.728,E2 -13638.728} C_VEL
LIN {X 0,Y 353.529,Z 467.246,A -85,B 0,C 180,E1 -13639.929,E2 -13639.929} C_VEL
LIN {X 0,Y 354.579,Z 455.84,A -85,B 0,C 180,E1 -13640.951,E2 -13640.951} C_VEL
LIN {X 0,Y 355.583,Z 443.757,A -85,B 0,C 180,E1 -13641.77,E2 -13641.77} C_VEL
LIN {X 0,Y 356.217,Z 430.494,A -85,B 0,C 180,E1 -13642.417,E2 -13642.417} C_VEL
LIN {X 0,Y 356.801,Z 417.101,A -85,B 0,C 180,E1 -13642.815,E2 -13642.815} C_VEL
LIN {X 0,Y 358.493,Z 342.127,A -85,B 0,C 180,E1 -13644.408,E2 -13644.408} C_VEL
LIN {X 0,Y 355.846,Z 330.29,A -85,B 0,C 180,E1 -13644.885,E2 -13644.885} C_VEL
LIN {X 0,Y 349.7,Z 315.268,A -85,B 0,C 180,E1 -13645.756,E2 -13645.756} C_VEL
LIN {X 0,Y 347.715,Z 307.175,A -85,B 0,C 180,E1 -13648.044,E2 -13648.044} C_VEL
LIN {X 0,Y 347.767,Z 307.168,A -85,B 0,C 180,E1 -13650.986,E2 -13650.986} C_VEL
LIN {X 0,Y 347.791,Z 307.169,A -85,B 0,C 180,E1 -13653.604,E2 -13653.604} C_VEL
LIN {X 0,Y 347.746,Z 307.176,A -85,B 0,C 180,E1 -13656.159,E2 -13656.159} C_VEL
LIN {X 0,Y 347.761,Z 307.17,A -85,B 0,C 180,E1 -13659.906,E2 -13659.906} C_VEL
LIN {X 0,Y 347.822,Z 307.162,A -85,B 0,C 180,E1 -13662.357,E2 -13662.357} C_VEL
LIN {X 0,Y 347.853,Z 307.155,A -85,B 0,C 180,E1 -13665.969,E2 -13665.969} C_VEL
LIN {X 0,Y 347.85,Z 307.15,A -85,B 0,C 180,E1 -13669.523,E2 -13669.523} C_VEL
LIN {X 0,Y 348.043,Z 307.128,A -85,B 0,C 180,E1 -13673.041,E2 -13673.041} C_VEL
LIN {X 0,Y 348.161,Z 307.114,A -85,B 0,C 180,E1 -13677.686,E2 -13677.686} C_VEL
LIN {X 0,Y 348.278,Z 307.092,A -85,B 0,C 180,E1 -13680,E2 -13680} C_VEL
LIN {X 0,Y 348.161,Z 307.115,A -85,B 0,C 180,E1 -13682.314,E2 -13682.314} C_VEL
LIN {X 0,Y 348.046,Z 307.126,A -85,B 0,C 180,E1 -13686.959,E2 -13686.959} C_VEL
LIN {X 0,Y 347.887,Z 307.15,A -85,B 0,C 180,E1 -13690.476,E2 -13690.476} C_VEL
LIN {X 0,Y 347.854,Z 307.152,A -85,B 0,C 180,E1 -13694.152,E2 -13694.152} C_VEL
LIN {X 0,Y 347.849,Z 307.151,A -85,B 0,C 180,E1 -13698.293,E2 -13698.293} C_VEL
LIN {X 0,Y 347.781,Z 307.161,A -85,B 0,C 180,E1 -13701.652,E2 -13701.652} C_VEL
LIN {X 0,Y 347.78,Z 307.155,A -85,B 0,C 180,E1 -13705.111,E2 -13705.111} C_VEL
LIN {X 0,Y 347.772,Z 307.157,A -85,B 0,C 180,E1 -13707.697,E2 -13707.697} C_VEL
LIN {X 0,Y 347.726,Z 307.168,A -85,B 0,C 180,E1 -13710.35,E2 -13710.35} C_VEL
LIN {X 0,Y 347.711,Z 307.169,A -85,B 0,C 180,E1 -13714.468,E2 -13714.468} C_VEL
LIN {X 0,Y 347.804,Z 307.158,A -85,B 0,C 180,E1 -13718.006,E2 -13718.006} C_VEL
LIN {X 0,Y 347.754,Z 307.17,A -85,B 0,C 180,E1 -13721.83,E2 -13721.83} C_VEL
LIN {X 0,Y 347.803,Z 307.166,A -85,B 0,C 180,E1 -13725.011,E2 -13725.011} C_VEL
LIN {X 0,Y 347.759,Z 307.169,A -85,B 0,C 180,E1 -13728.396,E2 -13728.396} C_VEL
LIN {X 0,Y 347.754,Z 307.168,A -85,B 0,C 180,E1 -13732.016,E2 -13732.016} C_VEL
LIN {X 0,Y 347.725,Z 307.176,A -85,B 0,C 180,E1 -13735.541,E2 -13735.541} C_VEL
LIN {X 0,Y 347.754,Z 307.246,A -85,B 0,C 180,E1 -13738.648,E2 -13738.648} C_VEL
LIN {X 0,Y 350.485,Z 318.512,A -85,B 0,C 180,E1 -13741.707,E2 -13741.707} C_VEL
LIN {X 0,Y 352.347,Z 328.625,A -85,B 0,C 180,E1 -13744.295,E2 -13744.295} C_VEL
LIN {X 0,Y 351.388,Z 338.051,A -85,B 0,C 180,E1 -13746.446,E2 -13746.446} C_VEL
LIN {X 0,Y 355.865,Z 362.01,A -85,B 0,C 180,E1 -13747.359,E2 -13747.359} C_VEL
LIN {X 0,Y 357.847,Z 376.7,A -85,B 0,C 180,E1 -13747.844,E2 -13747.844} C_VEL
LIN {X 0,Y 356.199,Z 447.1,A -85,B 0,C 180,E1 -13749.354,E2 -13749.354} C_VEL
LIN {X 0,Y 355.441,Z 460.897,A -85,B 0,C 180,E1 -13749.874,E2 -13749.874} C_VEL
LIN {X 0,Y 354.334,Z 473.91,A -85,B 0,C 180,E1 -13750.601,E2 -13750.601} C_VEL
LIN {X 0,Y 353.093,Z 486.528,A -85,B 0,C 180,E1 -13751.585,E2 -13751.585} C_VEL
LIN {X 0,Y 351.843,Z 497.8,A -85,B 0,C 180,E1 -13752.72,E2 -13752.72} C_VEL
LIN {X 0,Y 350.661,Z 507.6,A -85,B 0,C 180,E1 -13753.951,E2 -13753.951} C_VEL
LIN {X 0,Y 349.445,Z 517.185,A -85,B 0,C 180,E1 -13755.445,E2 -13755.445} C_VEL
LIN {X 0,Y 348.321,Z 526.171,A -85,B 0,C 180,E1 -13757.181,E2 -13757.181} C_VEL
LIN {X 0,Y 347.411,Z 533.416,A -85,B 0,C 180,E1 -13758.924,E2 -13758.924} C_VEL
LIN {X 0,Y 346.836,Z 539.21,A -85,B 0,C 180,E1 -13760.675,E2 -13760.675} C_VEL
LIN {X 0,Y 346.46,Z 543.787,A -85,B 0,C 180,E1 -13762.428,E2 -13762.428} C_VEL
LIN {X 0,Y 346.198,Z 547.278,A -85,B 0,C 180,E1 -13764.179,E2 -13764.179} C_VEL
LIN {X 0,Y 346.173,Z 549.025,A -85,B 0,C 180,E1 -13765.346,E2 -13765.346} C_VEL
LIN {X 0,Y 346.147,Z 550.364,A -85,B 0,C 180,E1 -13766.512,E2 -13766.512} C_VEL
LIN {X 0,Y 346.112,Z 551.304,A -85,B 0,C 180,E1 -13767.676,E2 -13767.676} C_VEL
LIN {X 0,Y 346.17,Z 551.819,A -85,B 0,C 180,E1 -13768.841,E2 -13768.841} C_VEL
LIN {X 0,Y 346.234,Z 551.913,A -85,B 0,C 180,E1 -13770.004,E2 -13770.004} C_VEL
LIN {X 0,Y 346.187,Z 551.61,A -85,B 0,C 180,E1 -13771.167,E2 -13771.167} C_VEL
LIN {X 0,Y 346.117,Z 550.912,A -85,B 0,C 180,E1 -13772.331,E2 -13772.331} C_VEL
LIN {X 0,Y 346.15,Z 549.786,A -85,B 0,C 180,E1 -13773.496,E2 -13773.496} C_VEL
LIN {X 0,Y 346.194,Z 548.216,A -85,B 0,C 180,E1 -13774.661,E2 -13774.661} C_VEL
LIN {X 0,Y 346.247,Z 545.044,A -85,B 0,C 180,E1 -13776.412,E2 -13776.412} C_VEL
LIN {X 0,Y 346.522,Z 540.789,A -85,B 0,C 180,E1 -13778.165,E2 -13778.165} C_VEL
LIN {X 0,Y 347.027,Z 534.31,A -85,B 0,C 180,E1 -13780.21,E2 -13780.21} C_VEL
LIN {X 0,Y 347.699,Z 527.214,A -85,B 0,C 180,E1 -13781.96,E2 -13781.96} C_VEL
LIN {X 0,Y 348.649,Z 518.327,A -85,B 0,C 180,E1 -13783.704,E2 -13783.704} C_VEL
LIN {X 0,Y 349.655,Z 509.221,A -85,B 0,C 180,E1 -13785.15,E2 -13785.15} C_VEL
LIN {X 0,Y 350.614,Z 499.174,A -85,B 0,C 180,E1 -13786.45,E2 -13786.45} C_VEL
LIN {X 0,Y 351.773,Z 488.02,A -85,B 0,C 180,E1 -13787.591,E2 -13787.591} C_VEL
LIN {X 0,Y 352.877,Z 475.532,A -85,B 0,C 180,E1 -13788.585,E2 -13788.585} C_VEL
LIN {X 0,Y 353.819,Z 462.882,A -85,B 0,C 180,E1 -13789.323,E2 -13789.323} C_VEL
LIN {X 0,Y 354.519,Z 449.556,A -85,B 0,C 180,E1 -13789.848,E2 -13789.848} C_VEL
LIN {X 0,Y 355.319,Z 417.401,A -85,B 0,C 180,E1 -13790.556,E2 -13790.556} C_VEL
LIN {X 0,Y 355.915,Z 374.589,A -85,B 0,C 180,E1 -13791.465,E2 -13791.465} C_VEL
LIN {X 0,Y 350.626,Z 339.534,A -85,B 0,C 180,E1 -13792.559,E2 -13792.559} C_VEL
LIN {X 0,Y 351.797,Z 327.391,A -85,B 0,C 180,E1 -13795.409,E2 -13795.409} C_VEL
LIN {X 0,Y 350.421,Z 319.314,A -85,B 0,C 180,E1 -13797.472,E2 -13797.472} C_VEL
LIN {X 0,Y 347.79,Z 307.164,A -85,B 0,C 180,E1 -13800.724,E2 -13800.724} C_VEL
LIN {X 0,Y 347.75,Z 307.167,A -85,B 0,C 180,E1 -13804.465,E2 -13804.465} C_VEL
LIN {X 0,Y 347.777,Z 307.164,A -85,B 0,C 180,E1 -13807.989,E2 -13807.989} C_VEL
LIN {X 0,Y 347.755,Z 307.165,A -85,B 0,C 180,E1 -13811.831,E2 -13811.831} C_VEL
LIN {X 0,Y 347.708,Z 307.17,A -85,B 0,C 180,E1 -13815.028,E2 -13815.028} C_VEL
LIN {X 0,Y 347.753,Z 307.169,A -85,B 0,C 180,E1 -13818.398,E2 -13818.398} C_VEL
LIN {X 0,Y 347.776,Z 307.162,A -85,B 0,C 180,E1 -13822.012,E2 -13822.012} C_VEL
LIN {X 0,Y 347.746,Z 307.164,A -85,B 0,C 180,E1 -13825.536,E2 -13825.536} C_VEL
LIN {X 0,Y 347.746,Z 307.167,A -85,B 0,C 180,E1 -13828.3,E2 -13828.3} C_VEL
LIN {X 0,Y 347.779,Z 307.165,A -85,B 0,C 180,E1 -13830.988,E2 -13830.988} C_VEL
LIN {X 0,Y 347.83,Z 307.154,A -85,B 0,C 180,E1 -13833.608,E2 -13833.608} C_VEL
LIN {X 0,Y 347.786,Z 307.16,A -85,B 0,C 180,E1 -13836.162,E2 -13836.162} C_VEL
LIN {X 0,Y 347.784,Z 307.16,A -85,B 0,C 180,E1 -13839.908,E2 -13839.908} C_VEL
LIN {X 0,Y 347.829,Z 307.156,A -85,B 0,C 180,E1 -13843.568,E2 -13843.568} C_VEL
LIN {X 0,Y 347.886,Z 307.153,A -85,B 0,C 180,E1 -13847.16,E2 -13847.16} C_VEL
LIN {X 0,Y 348.042,Z 307.13,A -85,B 0,C 180,E1 -13851.67,E2 -13851.67} C_VEL
LIN {X 0,Y 348.057,Z 307.126,A -85,B 0,C 180,E1 -13854.206,E2 -13854.206} C_VEL
LIN {X 0,Y 348.199,Z 307.112,A -85,B 0,C 180,E1 -13857.686,E2 -13857.686} C_VEL
LIN {X 0,Y 348.28,Z 307.099,A -85,B 0,C 180,E1 -13860,E2 -13860} C_VEL
LIN {X 0,Y 348.199,Z 307.108,A -85,B 0,C 180,E1 -13862.314,E2 -13862.314} C_VEL
LIN {X 0,Y 348.051,Z 307.127,A -85,B 0,C 180,E1 -13866.959,E2 -13866.959} C_VEL
LIN {X 0,Y 347.892,Z 307.147,A -85,B 0,C 180,E1 -13870.476,E2 -13870.476} C_VEL
LIN {X 0,Y 347.899,Z 307.148,A -85,B 0,C 180,E1 -13874.15,E2 -13874.15} C_VEL
LIN {X 0,Y 347.828,Z 307.157,A -85,B 0,C 180,E1 -13878.259,E2 -13878.259} C_VEL
LIN {X 0,Y 347.762,Z 307.165,A -85,B 0,C 180,E1 -13881.624,E2 -13881.624} C_VEL
LIN {X 0,Y 347.732,Z 307.166,A -85,B 0,C 180,E1 -13885.115,E2 -13885.115} C_VEL
LIN {X 0,Y 347.724,Z 307.169,A -85,B 0,C 180,E1 -13887.701,E2 -13887.701} C_VEL
LIN {X 0,Y 347.727,Z 307.172,A -85,B 0,C 180,E1 -13890.35,E2 -13890.35} C_VEL
LIN {X 0,Y 347.75,Z 307.168,A -85,B 0,C 180,E1 -13894.043,E2 -13894.043} C_VEL
LIN {X 0,Y 347.755,Z 307.163,A -85,B 0,C 180,E1 -13897.322,E2 -13897.322} C_VEL
LIN {X 0,Y 347.698,Z 307.175,A -85,B 0,C 180,E1 -13900.302,E2 -13900.302} C_VEL
LIN {X 0,Y 347.72,Z 307.168,A -85,B 0,C 180,E1 -13903.409,E2 -13903.409} C_VEL
LIN {X 0,Y 347.715,Z 307.174,A -85,B 0,C 180,E1 -13906.688,E2 -13906.688} C_VEL
LIN {X 0,Y 347.705,Z 307.171,A -85,B 0,C 180,E1 -13910.182,E2 -13910.182} C_VEL
LIN {X 0,Y 347.742,Z 307.171,A -85,B 0,C 180,E1 -13912.675,E2 -13912.675} C_VEL
LIN {X 0,Y 347.73,Z 307.166,A -85,B 0,C 180,E1 -13915.961,E2 -13915.961} C_VEL
LIN {X 0,Y 347.733,Z 307.166,A -85,B 0,C 180,E1 -13919.649,E2 -13919.649} C_VEL
LIN {X 0,Y 347.743,Z 307.166,A -85,B 0,C 180,E1 -13923.598,E2 -13923.598} C_VEL
LIN {X 0,Y 347.768,Z 307.162,A -85,B 0,C 180,E1 -13926.158,E2 -13926.158} C_VEL
LIN {X 0,Y 347.806,Z 307.157,A -85,B 0,C 180,E1 -13929.906,E2 -13929.906} C_VEL
LIN {X 0,Y 347.837,Z 307.156,A -85,B 0,C 180,E1 -13933.566,E2 -13933.566} C_VEL
LIN {X 0,Y 347.895,Z 307.151,A -85,B 0,C 180,E1 -13937.158,E2 -13937.158} C_VEL
LIN {X 0,Y 347.939,Z 307.141,A -85,B 0,C 180,E1 -13940.698,E2 -13940.698} C_VEL
LIN {X 0,Y 348.04,Z 307.128,A -85,B 0,C 180,E1 -13944.202,E2 -13944.202} C_VEL
LIN {X 0,Y 348.19,Z 307.114,A -85,B 0,C 180,E1 -13947.683,E2 -13947.683} C_VEL
LIN {X 0,Y 348.118,Z 307.12,A -85,B 0,C 180,E1 -13951.153,E2 -13951.153} C_VEL
LIN {X 0,Y 348.191,Z 307.11,A -85,B 0,C 180,E1 -13952.31,E2 -13952.31} C_VEL
LIN {X 0,Y 348.045,Z 307.131,A -85,B 0,C 180,E1 -13956.955,E2 -13956.955} C_VEL
LIN {X 0,Y 348.036,Z 307.332,A -85,B 0,C 180,E1 -13957.173,E2 -13957.173} C_VEL
LIN {X 0,Y 349.515,Z 315.17,A -85,B 0,C 180,E1 -13959.435,E2 -13959.435} C_VEL
LIN {X 0,Y 353.87,Z 328.161,A -85,B 0,C 180,E1 -13960.003,E2 -13960.003} C_VEL
LIN {X 0,Y 356.533,Z 342.065,A -85,B 0,C 180,E1 -13960.47,E2 -13960.47} C_VEL
LIN {X 0,Y 354.812,Z 422.814,A -85,B 0,C 180,E1 -13962.181,E2 -13962.181} C_VEL
LIN {X 0,Y 354.234,Z 436.896,A -85,B 0,C 180,E1 -13962.73,E2 -13962.73} C_VEL
LIN {X 0,Y 353.527,Z 449.202,A -85,B 0,C 180,E1 -13963.443,E2 -13963.443} C_VEL
LIN {X 0,Y 352.56,Z 461.652,A -85,B 0,C 180,E1 -13964.424,E2 -13964.424} C_VEL
LIN {X 0,Y 351.497,Z 473.471,A -85,B 0,C 180,E1 -13965.629,E2 -13965.629} C_VEL
LIN {X 0,Y 350.308,Z 484.431,A -85,B 0,C 180,E1 -13967.057,E2 -13967.057} C_VEL
LIN {X 0,Y 349.413,Z 493.135,A -85,B 0,C 180,E1 -13968.464,E2 -13968.464} C_VEL
LIN {X 0,Y 348.57,Z 501.122,A -85,B 0,C 180,E1 -13970.04,E2 -13970.04} C_VEL
LIN {X 0,Y 347.8,Z 507.736,A -85,B 0,C 180,E1 -13971.639,E2 -13971.639} C_VEL
LIN {X 0,Y 347.294,Z 513.086,A -85,B 0,C 180,E1 -13973.236,E2 -13973.236} C_VEL
LIN {X 0,Y 346.797,Z 518.212,A -85,B 0,C 180,E1 -13975.181,E2 -13975.181} C_VEL
LIN {X 0,Y 346.435,Z 521.44,A -85,B 0,C 180,E1 -13976.796,E2 -13976.796} C_VEL
LIN {X 0,Y 346.21,Z 523.18,A -85,B 0,C 180,E1 -13977.949,E2 -13977.949} C_VEL
LIN {X 0,Y 346.093,Z 524.596,A -85,B 0,C 180,E1 -13979.168,E2 -13979.168} C_VEL
LIN {X 0,Y 345.962,Z 526.058,A -85,B 0,C 180,E1 -13981.438,E2 -13981.438} C_VEL
LIN {X 0,Y 345.985,Z 526.114,A -85,B 0,C 180,E1 -13982.988,E2 -13982.988} C_VEL
LIN {X 0,Y 345.388,Z 525.928,A -85,B 0,C 180,E1 -13983.96,E2 -13983.96} C_VEL
LIN {X 0,Y 342.657,Z 524.965,A -85,B 0,C 180,E1 -13985.539,E2 -13985.539} C_VEL
LIN {X 0,Y 340.401,Z 523.751,A -85,B 0,C 180,E1 -13986.808,E2 -13986.808} C_VEL
LIN {X 0,Y 339.552,Z 522.479,A -85,B 0,C 180,E1 -13987.778,E2 -13987.778} C_VEL
LIN {X 0,Y 339.549,Z 521.985,A -85,B 0,C 180,E1 -13988.104,E2 -13988.104} C_VEL
LIN {X 0,Y 340.081,Z 518.031,A -85,B 0,C 180,E1 -13990.126,E2 -13990.126} C_VEL
LIN {X 0,Y 340.8,Z 512.898,A -85,B 0,C 180,E1 -13992.064,E2 -13992.064} C_VEL
LIN {X 0,Y 341.691,Z 506.461,A -85,B 0,C 180,E1 -13993.954,E2 -13993.954} C_VEL
LIN {X 0,Y 342.89,Z 498.333,A -85,B 0,C 180,E1 -13995.828,E2 -13995.828} C_VEL
LIN {X 0,Y 344.028,Z 490.206,A -85,B 0,C 180,E1 -13997.333,E2 -13997.333} C_VEL
LIN {X 0,Y 345.363,Z 480.228,A -85,B 0,C 180,E1 -13998.835,E2 -13998.835} C_VEL
LIN {X 0,Y 346.603,Z 469.941,A -85,B 0,C 180,E1 -14000.08,E2 -14000.08} C_VEL
LIN {X 0,Y 347.807,Z 458.009,A -85,B 0,C 180,E1 -14001.214,E2 -14001.214} C_VEL
LIN {X 0,Y 348.91,Z 445.594,A -85,B 0,C 180,E1 -14002.111,E2 -14002.111} C_VEL
LIN {X 0,Y 349.627,Z 433.5,A -85,B 0,C 180,E1 -14002.751,E2 -14002.751} C_VEL
LIN {X 0,Y 350.214,Z 419.935,A -85,B 0,C 180,E1 -14003.207,E2 -14003.207} C_VEL
LIN {X 0,Y 352.027,Z 342.989,A -85,B 0,C 180,E1 -14004.883,E2 -14004.883} C_VEL
LIN {X 0,Y 349.757,Z 332.898,A -85,B 0,C 180,E1 -14005.303,E2 -14005.303} C_VEL
LIN {X 0,Y 343.275,Z 317.476,A -85,B 0,C 180,E1 -14006.222,E2 -14006.222} C_VEL
LIN {X 0,Y 342.526,Z 315.58,A -85,B 0,C 180,E1 -14006.359,E2 -14006.359} C_VEL
LIN {X 0,Y 340.667,Z 308.051,A -85,B 0,C 180,E1 -14008.52,E2 -14008.52} C_VEL
LIN {X 0,Y 340.702,Z 308.049,A -85,B 0,C 180,E1 -14011.677,E2 -14011.677} C_VEL
LIN {X 0,Y 340.732,Z 308.049,A -85,B 0,C 180,E1 -14014.332,E2 -14014.332} C_VEL
LIN {X 0,Y 340.7,Z 308.053,A -85,B 0,C 180,E1 -14018.204,E2 -14018.204} C_VEL
LIN {X 0,Y 340.814,Z 308.032,A -85,B 0,C 180,E1 -14021.982,E2 -14021.982} C_VEL
LIN {X 0,Y 340.808,Z 308.032,A -85,B 0,C 180,E1 -14025.715,E2 -14025.715} C_VEL
LIN {X 0,Y 340.802,Z 308.028,A -85,B 0,C 180,E1 -14029.304,E2 -14029.304} C_VEL
LIN {X 0,Y 341.012,Z 308.003,A -85,B 0,C 180,E1 -14032.897,E2 -14032.897} C_VEL
LIN {X 0,Y 341.123,Z 307.991,A -85,B 0,C 180,E1 -14037.638,E2 -14037.638} C_VEL
LIN {X 0,Y 341.229,Z 307.97,A -85,B 0,C 180,E1 -14040,E2 -14040} C_VEL
LIN {X 0,Y 341.124,Z 307.992,A -85,B 0,C 180,E1 -14042.362,E2 -14042.362} C_VEL
LIN {X 0,Y 341.014,Z 308.001,A -85,B 0,C 180,E1 -14047.103,E2 -14047.103} C_VEL
LIN {X 0,Y 340.829,Z 308.031,A -85,B 0,C 180,E1 -14050.695,E2 -14050.695} C_VEL
LIN {X 0,Y 340.819,Z 308.029,A -85,B 0,C 180,E1 -14054.327,E2 -14054.327} C_VEL
LIN {X 0,Y 340.796,Z 308.03,A -85,B 0,C 180,E1 -14058.469,E2 -14058.469} C_VEL
LIN {X 0,Y 340.721,Z 308.039,A -85,B 0,C 180,E1 -14061.863,E2 -14061.863} C_VEL
LIN {X 0,Y 340.736,Z 308.039,A -85,B 0,C 180,E1 -14065.667,E2 -14065.667} C_VEL
LIN {X 0,Y 340.702,Z 308.036,A -85,B 0,C 180,E1 -14068.323,E2 -14068.323} C_VEL
LIN {X 0,Y 340.666,Z 308.049,A -85,B 0,C 180,E1 -14071.048,E2 -14071.048} C_VEL
LIN {X 0,Y 340.694,Z 308.043,A -85,B 0,C 180,E1 -14075.282,E2 -14075.282} C_VEL
LIN {X 0,Y 340.743,Z 308.037,A -85,B 0,C 180,E1 -14078.404,E2 -14078.404} C_VEL
LIN {X 0,Y 340.722,Z 308.048,A -85,B 0,C 180,E1 -14082.06,E2 -14082.06} C_VEL
LIN {X 0,Y 340.754,Z 308.045,A -85,B 0,C 180,E1 -14085.482,E2 -14085.482} C_VEL
LIN {X 0,Y 340.701,Z 308.048,A -85,B 0,C 180,E1 -14088.701,E2 -14088.701} C_VEL
LIN {X 0,Y 340.717,Z 308.045,A -85,B 0,C 180,E1 -14091.779,E2 -14091.779} C_VEL
LIN {X 0,Y 340.703,Z 308.05,A -85,B 0,C 180,E1 -14095.601,E2 -14095.601} C_VEL
LIN {X 0,Y 340.685,Z 308.115,A -85,B 0,C 180,E1 -14098.142,E2 -14098.142} C_VEL
LIN {X 0,Y 343.084,Z 317.756,A -85,B 0,C 180,E1 -14100.855,E2 -14100.855} C_VEL
LIN {X 0,Y 345.339,Z 329.034,A -85,B 0,C 180,E1 -14103.838,E2 -14103.838} C_VEL
LIN {X 0,Y 345.296,Z 332.614,A -85,B 0,C 180,E1 -14104.702,E2 -14104.702} C_VEL
LIN {X 0,Y 344.701,Z 337.787,A -85,B 0,C 180,E1 -14105.901,E2 -14105.901} C_VEL
LIN {X 0,Y 349.255,Z 361.839,A -85,B 0,C 180,E1 -14106.851,E2 -14106.851} C_VEL
LIN {X 0,Y 351.371,Z 377.267,A -85,B 0,C 180,E1 -14107.377,E2 -14107.377} C_VEL
LIN {X 0,Y 349.665,Z 447.151,A -85,B 0,C 180,E1 -14108.911,E2 -14108.911} C_VEL
LIN {X 0,Y 348.883,Z 460.807,A -85,B 0,C 180,E1 -14109.441,E2 -14109.441} C_VEL
LIN {X 0,Y 347.75,Z 473.211,A -85,B 0,C 180,E1 -14110.142,E2 -14110.142} C_VEL
LIN {X 0,Y 346.565,Z 485.126,A -85,B 0,C 180,E1 -14111.072,E2 -14111.072} C_VEL
LIN {X 0,Y 345.181,Z 496.584,A -85,B 0,C 180,E1 -14112.223,E2 -14112.223} C_VEL
LIN {X 0,Y 343.891,Z 507.238,A -85,B 0,C 180,E1 -14113.572,E2 -14113.572} C_VEL
LIN {X 0,Y 342.56,Z 517.135,A -85,B 0,C 180,E1 -14115.145,E2 -14115.145} C_VEL
LIN {X 0,Y 341.376,Z 526.087,A -85,B 0,C 180,E1 -14116.916,E2 -14116.916} C_VEL
LIN {X 0,Y 340.408,Z 533.292,A -85,B 0,C 180,E1 -14118.694,E2 -14118.694} C_VEL
LIN {X 0,Y 339.79,Z 539.053,A -85,B 0,C 180,E1 -14120.48,E2 -14120.48} C_VEL
LIN {X 0,Y 339.391,Z 543.606,A -85,B 0,C 180,E1 -14122.269,E2 -14122.269} C_VEL
LIN {X 0,Y 339.13,Z 547.17,A -85,B 0,C 180,E1 -14124.119,E2 -14124.119} C_VEL
LIN {X 0,Y 339.071,Z 550.136,A -85,B 0,C 180,E1 -14126.439,E2 -14126.439} C_VEL
LIN {X 0,Y 339.024,Z 551.064,A -85,B 0,C 180,E1 -14127.628,E2 -14127.628} C_VEL
LIN {X 0,Y 339.071,Z 551.558,A -85,B 0,C 180,E1 -14128.816,E2 -14128.816} C_VEL
LIN {X 0,Y 339.139,Z 551.642,A -85,B 0,C 180,E1 -14130.004,E2 -14130.004} C_VEL
LIN {X 0,Y 339.088,Z 551.328,A -85,B 0,C 180,E1 -14131.191,E2 -14131.191} C_VEL
LIN {X 0,Y 339.029,Z 550.621,A -85,B 0,C 180,E1 -14132.38,E2 -14132.38} C_VEL
LIN {X 0,Y 339.075,Z 549.473,A -85,B 0,C 180,E1 -14133.569,E2 -14133.569} C_VEL
LIN {X 0,Y 339.092,Z 547.89,A -85,B 0,C 180,E1 -14134.759,E2 -14134.759} C_VEL
LIN {X 0,Y 339.17,Z 544.692,A -85,B 0,C 180,E1 -14136.547,E2 -14136.547} C_VEL
LIN {X 0,Y 339.459,Z 540.41,A -85,B 0,C 180,E1 -14138.336,E2 -14138.336} C_VEL
LIN {X 0,Y 340.007,Z 533.899,A -85,B 0,C 180,E1 -14140.423,E2 -14140.423} C_VEL
LIN {X 0,Y 340.733,Z 526.747,A -85,B 0,C 180,E1 -14142.209,E2 -14142.209} C_VEL
LIN {X 0,Y 341.715,Z 517.812,A -85,B 0,C 180,E1 -14143.988,E2 -14143.988} C_VEL
LIN {X 0,Y 342.767,Z 508.467,A -85,B 0,C 180,E1 -14145.49,E2 -14145.49} C_VEL
LIN {X 0,Y 343.8,Z 498.501,A -85,B 0,C 180,E1 -14146.786,E2 -14146.786} C_VEL
LIN {X 0,Y 345.005,Z 487.241,A -85,B 0,C 180,E1 -14147.948,E2 -14147.948} C_VEL
LIN {X 0,Y 346.127,Z 474.61,A -85,B 0,C 180,E1 -14148.961,E2 -14148.961} C_VEL
LIN {X 0,Y 347.115,Z 461.618,A -85,B 0,C 180,E1 -14149.711,E2 -14149.711} C_VEL
LIN {X 0,Y 347.768,Z 448.925,A -85,B 0,C 180,E1 -14150.212,E2 -14150.212} C_VEL
LIN {X 0,Y 348.835,Z 404.606,A -85,B 0,C 180,E1 -14151.188,E2 -14151.188} C_VEL
LIN {X 0,Y 349.273,Z 375.828,A -85,B 0,C 180,E1 -14151.81,E2 -14151.81} C_VEL
LIN {X 0,Y 343.763,Z 339.241,A -85,B 0,C 180,E1 -14152.997,E2 -14152.997} C_VEL
LIN {X 0,Y 344.829,Z 329.419,A -85,B 0,C 180,E1 -14155.343,E2 -14155.343} C_VEL
LIN {X 0,Y 343.937,Z 322.801,A -85,B 0,C 180,E1 -14157.045,E2 -14157.045} C_VEL
LIN {X 0,Y 341.211,Z 310.032,A -85,B 0,C 180,E1 -14160.501,E2 -14160.501} C_VEL
LIN {X 0,Y 340.744,Z 308.04,A -85,B 0,C 180,E1 -14161.128,E2 -14161.128} C_VEL
LIN {X 0,Y 340.723,Z 308.039,A -85,B 0,C 180,E1 -14165.28,E2 -14165.28} C_VEL
LIN {X 0,Y 340.714,Z 308.045,A -85,B 0,C 180,E1 -14168.387,E2 -14168.387} C_VEL
LIN {X 0,Y 340.703,Z 308.045,A -85,B 0,C 180,E1 -14172.046,E2 -14172.046} C_VEL
LIN {X 0,Y 340.656,Z 308.052,A -85,B 0,C 180,E1 -14176.228,E2 -14176.228} C_VEL
LIN {X 0,Y 340.691,Z 308.044,A -85,B 0,C 180,E1 -14179.754,E2 -14179.754} C_VEL
LIN {X 0,Y 340.707,Z 308.042,A -85,B 0,C 180,E1 -14183.259,E2 -14183.259} C_VEL
LIN {X 0,Y 340.695,Z 308.044,A -85,B 0,C 180,E1 -14186.154,E2 -14186.154} C_VEL
LIN {X 0,Y 340.739,Z 308.039,A -85,B 0,C 180,E1 -14190.329,E2 -14190.329} C_VEL
LIN {X 0,Y 340.804,Z 308.034,A -85,B 0,C 180,E1 -14193.02,E2 -14193.02} C_VEL
LIN {X 0,Y 340.755,Z 308.036,A -85,B 0,C 180,E1 -14195.638,E2 -14195.638} C_VEL
LIN {X 0,Y 340.72,Z 308.041,A -85,B 0,C 180,E1 -14199.472,E2 -14199.472} C_VEL
LIN {X 0,Y 340.791,Z 308.031,A -85,B 0,C 180,E1 -14201.981,E2 -14201.981} C_VEL
LIN {X 0,Y 340.853,Z 308.024,A -85,B 0,C 180,E1 -14205.716,E2 -14205.716} C_VEL
LIN {X 0,Y 340.846,Z 308.03,A -85,B 0,C 180,E1 -14209.305,E2 -14209.305} C_VEL
LIN {X 0,Y 341.056,Z 308,A -85,B 0,C 180,E1 -14212.898,E2 -14212.898} C_VEL
LIN {X 0,Y 341.161,Z 307.989,A -85,B 0,C 180,E1 -14217.639,E2 -14217.639} C_VEL
LIN {X 0,Y 341.232,Z 307.977,A -85,B 0,C 180,E1 -14220,E2 -14220} C_VEL
LIN {X 0,Y 341.161,Z 307.985,A -85,B 0,C 180,E1 -14222.361,E2 -14222.361} C_VEL
LIN {X 0,Y 340.999,Z 308.006,A -85,B 0,C 180,E1 -14227.103,E2 -14227.103} C_VEL
LIN {X 0,Y 340.844,Z 308.024,A -85,B 0,C 180,E1 -14230.695,E2 -14230.695} C_VEL
LIN {X 0,Y 340.864,Z 308.023,A -85,B 0,C 180,E1 -14234.325,E2 -14234.325} C_VEL
LIN {X 0,Y 340.785,Z 308.033,A -85,B 0,C 180,E1 -14238.44,E2 -14238.44} C_VEL
LIN {X 0,Y 340.719,Z 308.044,A -85,B 0,C 180,E1 -14241.842,E2 -14241.842} C_VEL
LIN {X 0,Y 340.704,Z 308.042,A -85,B 0,C 180,E1 -14244.82,E2 -14244.82} C_VEL
LIN {X 0,Y 340.672,Z 308.05,A -85,B 0,C 180,E1 -14248.326,E2 -14248.326} C_VEL
LIN {X 0,Y 340.682,Z 308.044,A -85,B 0,C 180,E1 -14251.046,E2 -14251.046} C_VEL
LIN {X 0,Y 340.716,Z 308.04,A -85,B 0,C 180,E1 -14255.279,E2 -14255.279} C_VEL
LIN {X 0,Y 340.695,Z 308.049,A -85,B 0,C 180,E1 -14258.382,E2 -14258.382} C_VEL
LIN {X 0,Y 340.67,Z 308.048,A -85,B 0,C 180,E1 -14262.039,E2 -14262.039} C_VEL
LIN {X 0,Y 340.63,Z 308.051,A -85,B 0,C 180,E1 -14265.451,E2 -14265.451} C_VEL
LIN {X 0,Y 340.648,Z 308.055,A -85,B 0,C 180,E1 -14268.683,E2 -14268.683} C_VEL
LIN {X 0,Y 340.715,Z 308.04,A -85,B 0,C 180,E1 -14271.769,E2 -14271.769} C_VEL
LIN {X 0,Y 340.705,Z 308.042,A -85,B 0,C 180,E1 -14275.6,E2 -14275.6} C_VEL
LIN {X 0,Y 340.682,Z 308.05,A -85,B 0,C 180,E1 -14278.952,E2 -14278.952} C_VEL
LIN {X 0,Y 340.691,Z 308.045,A -85,B 0,C 180,E1 -14282.503,E2 -14282.503} C_VEL
LIN {X 0,Y 340.745,Z 308.038,A -85,B 0,C 180,E1 -14285.635,E2 -14285.635} C_VEL
LIN {X 0,Y 340.736,Z 308.041,A -85,B 0,C 180,E1 -14289.471,E2 -14289.471} C_VEL
LIN {X 0,Y 340.799,Z 308.03,A -85,B 0,C 180,E1 -14291.978,E2 -14291.978} C_VEL
LIN {X 0,Y 340.876,Z 308.022,A -85,B 0,C 180,E1 -14295.702,E2 -14295.702} C_VEL
LIN {X 0,Y 340.851,Z 308.029,A -85,B 0,C 180,E1 -14299.302,E2 -14299.302} C_VEL
LIN {X 0,Y 341.004,Z 308.005,A -85,B 0,C 180,E1 -14302.893,E2 -14302.893} C_VEL
LIN {X 0,Y 340.813,Z 308.032,A -85,B 0,C 180,E1 -14305.265,E2 -14305.265} C_VEL
LIN {X 0,Y 341.127,Z 307.995,A -85,B 0,C 180,E1 -14307.635,E2 -14307.635} C_VEL
LIN {X 0,Y 341.089,Z 307.995,A -85,B 0,C 180,E1 -14311.177,E2 -14311.177} C_VEL
LIN {X 0,Y 341.128,Z 307.989,A -85,B 0,C 180,E1 -14312.358,E2 -14312.358} C_VEL
LIN {X 0,Y 341.02,Z 308.115,A -85,B 0,C 180,E1 -14316.838,E2 -14316.838} C_VEL
LIN {X 0,Y 342.365,Z 315.466,A -85,B 0,C 180,E1 -14319.001,E2 -14319.001} C_VEL
LIN {X 0,Y 347.534,Z 330.836,A -85,B 0,C 180,E1 -14319.682,E2 -14319.682} C_VEL
LIN {X 0,Y 349.858,Z 343.006,A -85,B 0,C 180,E1 -14320.101,E2 -14320.101} C_VEL
LIN {X 0,Y 348.079,Z 422.995,A -85,B 0,C 180,E1 -14321.829,E2 -14321.829} C_VEL
LIN {X 0,Y 347.488,Z 436.68,A -85,B 0,C 180,E1 -14322.367,E2 -14322.367} C_VEL
LIN {X 0,Y 346.72,Z 449.453,A -85,B 0,C 180,E1 -14323.115,E2 -14323.115} C_VEL
LIN {X 0,Y 345.86,Z 460.531,A -85,B 0,C 180,E1 -14323.99,E2 -14323.99} C_VEL
LIN {X 0,Y 344.702,Z 472.595,A -85,B 0,C 180,E1 -14325.214,E2 -14325.214} C_VEL
LIN {X 0,Y 343.639,Z 482.478,A -85,B 0,C 180,E1 -14326.473,E2 -14326.473} C_VEL
LIN {X 0,Y 342.677,Z 491.604,A -85,B 0,C 180,E1 -14327.912,E2 -14327.912} C_VEL
LIN {X 0,Y 341.705,Z 499.913,A -85,B 0,C 180,E1 -14329.52,E2 -14329.52} C_VEL
LIN {X 0,Y 340.926,Z 506.746,A -85,B 0,C 180,E1 -14331.141,E2 -14331.141} C_VEL
LIN {X 0,Y 340.258,Z 513.352,A -85,B 0,C 180,E1 -14333.101,E2 -14333.101} C_VEL
LIN {X 0,Y 339.735,Z 518.478,A -85,B 0,C 180,E1 -14335.085,E2 -14335.085} C_VEL
LIN {X 0,Y 339.284,Z 522.287,A -85,B 0,C 180,E1 -14337.104,E2 -14337.104} C_VEL
LIN {X 0,Y 338.971,Z 525.146,A -85,B 0,C 180,E1 -14339.448,E2 -14339.448} C_VEL
LIN {X 0,Y 338.89,Z 526.375,A -85,B 0,C 180,E1 -14341.759,E2 -14341.759} C_VEL
LIN {X 0,Y 338.955,Z 526.121,A -85,B 0,C 180,E1 -14344.036,E2 -14344.036} C_VEL
LIN {X 0,Y 339.206,Z 524.637,A -85,B 0,C 180,E1 -14346.095,E2 -14346.095} C_VEL
LIN {X 0,Y 339.549,Z 521.985,A -85,B 0,C 180,E1 -14348.104,E2 -14348.104} C_VEL
LIN {X 0,Y 339.129,Z 520.465,A -85,B 0,C 180,E1 -14349.065,E2 -14349.065} C_VEL
LIN {X 0,Y 336.703,Z 517.416,A -85,B 0,C 180,E1 -14350.612,E2 -14350.612} C_VEL
LIN {X 0,Y 334.379,Z 513.634,A -85,B 0,C 180,E1 -14352.134,E2 -14352.134} C_VEL
LIN {X 0,Y 334.132,Z 510.943,A -85,B 0,C 180,E1 -14353.04,E2 -14353.04} C_VEL
LIN {X 0,Y 335.153,Z 504.19,A -85,B 0,C 180,E1 -14354.899,E2 -14354.899} C_VEL
LIN {X 0,Y 336.376,Z 496.443,A -85,B 0,C 180,E1 -14356.605,E2 -14356.605} C_VEL
LIN {X 0,Y 337.727,Z 487.179,A -85,B 0,C 180,E1 -14358.248,E2 -14358.248} C_VEL
LIN {X 0,Y 338.974,Z 477.547,A -85,B 0,C 180,E1 -14359.625,E2 -14359.625} C_VEL
LIN {X 0,Y 340.396,Z 466.467,A -85,B 0,C 180,E1 -14360.89,E2 -14360.89} C_VEL
LIN {X 0,Y 341.639,Z 454.308,A -85,B 0,C 180,E1 -14361.973,E2 -14361.973} C_VEL
LIN {X 0,Y 342.619,Z 441.791,A -85,B 0,C 180,E1 -14362.807,E2 -14362.807} C_VEL
LIN {X 0,Y 343.301,Z 429.322,A -85,B 0,C 180,E1 -14363.4,E2 -14363.4} C_VEL
LIN {X 0,Y 343.877,Z 415.619,A -85,B 0,C 180,E1 -14363.786,E2 -14363.786} C_VEL
LIN {X 0,Y 345.584,Z 343.862,A -85,B 0,C 180,E1 -14365.378,E2 -14365.378} C_VEL
LIN {X 0,Y 343.698,Z 335.566,A -85,B 0,C 180,E1 -14365.739,E2 -14365.739} C_VEL
LIN {X 0,Y 337.537,Z 320.844,A -85,B 0,C 180,E1 -14366.645,E2 -14366.645} C_VEL
LIN {X 0,Y 335.358,Z 315.938,A -85,B 0,C 180,E1 -14366.984,E2 -14366.984} C_VEL
LIN {X 0,Y 333.643,Z 308.928,A -85,B 0,C 180,E1 -14369.062,E2 -14369.062} C_VEL
LIN {X 0,Y 333.704,Z 308.924,A -85,B 0,C 180,E1 -14372.397,E2 -14372.397} C_VEL
LIN {X 0,Y 333.686,Z 308.926,A -85,B 0,C 180,E1 -14375.087,E2 -14375.087} C_VEL
LIN {X 0,Y 333.631,Z 308.93,A -85,B 0,C 180,E1 -14379.016,E2 -14379.016} C_VEL
LIN {X 0,Y 333.75,Z 308.911,A -85,B 0,C 180,E1 -14381.587,E2 -14381.587} C_VEL
LIN {X 0,Y 333.765,Z 308.909,A -85,B 0,C 180,E1 -14385.575,E2 -14385.575} C_VEL
LIN {X 0,Y 333.771,Z 308.904,A -85,B 0,C 180,E1 -14389.076,E2 -14389.076} C_VEL
LIN {X 0,Y 333.959,Z 308.881,A -85,B 0,C 180,E1 -14392.746,E2 -14392.746} C_VEL
LIN {X 0,Y 333.764,Z 308.906,A -85,B 0,C 180,E1 -14395.168,E2 -14395.168} C_VEL
LIN {X 0,Y 334.06,Z 308.871,A -85,B 0,C 180,E1 -14397.588,E2 -14397.588} C_VEL
LIN {X 0,Y 334.181,Z 308.847,A -85,B 0,C 180,E1 -14400,E2 -14400} C_VEL
LIN {X 0,Y 334.061,Z 308.872,A -85,B 0,C 180,E1 -14402.411,E2 -14402.411} C_VEL
LIN {X 0,Y 333.969,Z 308.882,A -85,B 0,C 180,E1 -14406.04,E2 -14406.04} C_VEL
LIN {X 0,Y 333.926,Z 308.881,A -85,B 0,C 180,E1 -14408.486,E2 -14408.486} C_VEL
LIN {X 0,Y 333.75,Z 308.901,A -85,B 0,C 180,E1 -14412.156,E2 -14412.156} C_VEL
LIN {X 0,Y 333.734,Z 308.904,A -85,B 0,C 180,E1 -14415.888,E2 -14415.888} C_VEL
LIN {X 0,Y 333.713,Z 308.907,A -85,B 0,C 180,E1 -14419.692,E2 -14419.692} C_VEL
LIN {X 0,Y 333.659,Z 308.914,A -85,B 0,C 180,E1 -14423.591,E2 -14423.591} C_VEL
LIN {X 0,Y 333.698,Z 308.914,A -85,B 0,C 180,E1 -14426.25,E2 -14426.25} C_VEL
LIN {X 0,Y 333.673,Z 308.913,A -85,B 0,C 180,E1 -14428.976,E2 -14428.976} C_VEL
LIN {X 0,Y 333.607,Z 308.925,A -85,B 0,C 180,E1 -14432.591,E2 -14432.591} C_VEL
LIN {X 0,Y 333.679,Z 308.92,A -85,B 0,C 180,E1 -14436.139,E2 -14436.139} C_VEL
LIN {X 0,Y 333.685,Z 308.919,A -85,B 0,C 180,E1 -14439.187,E2 -14439.187} C_VEL
LIN {X 0,Y 333.674,Z 308.924,A -85,B 0,C 180,E1 -14442.518,E2 -14442.518} C_VEL
LIN {X 0,Y 333.702,Z 308.921,A -85,B 0,C 180,E1 -14445.982,E2 -14445.982} C_VEL
LIN {X 0,Y 333.678,Z 308.925,A -85,B 0,C 180,E1 -14449.31,E2 -14449.31} C_VEL
LIN {X 0,Y 333.644,Z 308.924,A -85,B 0,C 180,E1 -14453.173,E2 -14453.173} C_VEL
LIN {X 0,Y 333.618,Z 308.93,A -85,B 0,C 180,E1 -14456.797,E2 -14456.797} C_VEL
LIN {X 0,Y 333.627,Z 308.961,A -85,B 0,C 180,E1 -14457.598,E2 -14457.598} C_VEL
LIN {X 0,Y 336.206,Z 319.286,A -85,B 0,C 180,E1 -14460.585,E2 -14460.585} C_VEL
LIN {X 0,Y 338.42,Z 330.164,A -85,B 0,C 180,E1 -14463.545,E2 -14463.545} C_VEL
LIN {X 0,Y 338.452,Z 333.932,A -85,B 0,C 180,E1 -14464.483,E2 -14464.483} C_VEL
LIN {X 0,Y 338.069,Z 337.437,A -85,B 0,C 180,E1 -14465.315,E2 -14465.315} C_VEL
LIN {X 0,Y 342.894,Z 363.114,A -85,B 0,C 180,E1 -14466.372,E2 -14466.372} C_VEL
LIN {X 0,Y 344.923,Z 378.866,A -85,B 0,C 180,E1 -14466.918,E2 -14466.918} C_VEL
LIN {X 0,Y 343.137,Z 447.278,A -85,B 0,C 180,E1 -14468.451,E2 -14468.451} C_VEL
LIN {X 0,Y 342.296,Z 460.798,A -85,B 0,C 180,E1 -14468.987,E2 -14468.987} C_VEL
LIN {X 0,Y 341.108,Z 473.638,A -85,B 0,C 180,E1 -14469.739,E2 -14469.739} C_VEL
LIN {X 0,Y 339.872,Z 485.38,A -85,B 0,C 180,E1 -14470.685,E2 -14470.685} C_VEL
LIN {X 0,Y 338.439,Z 496.744,A -85,B 0,C 180,E1 -14471.856,E2 -14471.856} C_VEL
LIN {X 0,Y 337.104,Z 507.117,A -85,B 0,C 180,E1 -14473.205,E2 -14473.205} C_VEL
LIN {X 0,Y 335.696,Z 517.111,A -85,B 0,C 180,E1 -14474.834,E2 -14474.834} C_VEL
LIN {X 0,Y 334.446,Z 526.009,A -85,B 0,C 180,E1 -14476.64,E2 -14476.64} C_VEL
LIN {X 0,Y 333.396,Z 533.163,A -85,B 0,C 180,E1 -14478.453,E2 -14478.453} C_VEL
LIN {X 0,Y 332.761,Z 538.897,A -85,B 0,C 180,E1 -14480.277,E2 -14480.277} C_VEL
LIN {X 0,Y 332.328,Z 543.425,A -85,B 0,C 180,E1 -14482.104,E2 -14482.104} C_VEL
LIN {X 0,Y 332.032,Z 547.239,A -85,B 0,C 180,E1 -14484.174,E2 -14484.174} C_VEL
LIN {X 0,Y 331.996,Z 549.911,A -85,B 0,C 180,E1 -14486.363,E2 -14486.363} C_VEL
LIN {X 0,Y 331.94,Z 550.824,A -85,B 0,C 180,E1 -14487.577,E2 -14487.577} C_VEL
LIN {X 0,Y 331.974,Z 551.297,A -85,B 0,C 180,E1 -14488.791,E2 -14488.791} C_VEL
LIN {X 0,Y 332.043,Z 551.369,A -85,B 0,C 180,E1 -14490.004,E2 -14490.004} C_VEL
LIN {X 0,Y 331.99,Z 551.044,A -85,B 0,C 180,E1 -14491.217,E2 -14491.217} C_VEL
LIN {X 0,Y 331.944,Z 550.322,A -85,B 0,C 180,E1 -14492.431,E2 -14492.431} C_VEL
LIN {X 0,Y 332.001,Z 549.151,A -85,B 0,C 180,E1 -14493.645,E2 -14493.645} C_VEL
LIN {X 0,Y 332.015,Z 546.03,A -85,B 0,C 180,E1 -14495.796,E2 -14495.796} C_VEL
LIN {X 0,Y 332.309,Z 541.592,A -85,B 0,C 180,E1 -14497.905,E2 -14497.905} C_VEL
LIN {X 0,Y 332.766,Z 535.507,A -85,B 0,C 180,E1 -14500.038,E2 -14500.038} C_VEL
LIN {X 0,Y 333.419,Z 528.816,A -85,B 0,C 180,E1 -14501.863,E2 -14501.863} C_VEL
LIN {X 0,Y 334.456,Z 520.506,A -85,B 0,C 180,E1 -14503.677,E2 -14503.677} C_VEL
LIN {X 0,Y 335.482,Z 511.691,A -85,B 0,C 180,E1 -14505.231,E2 -14505.231} C_VEL
LIN {X 0,Y 336.538,Z 501.432,A -85,B 0,C 180,E1 -14506.69,E2 -14506.69} C_VEL
LIN {X 0,Y 337.862,Z 489.573,A -85,B 0,C 180,E1 -14508.027,E2 -14508.027} C_VEL
LIN {X 0,Y 339.029,Z 477.649,A -85,B 0,C 180,E1 -14509.059,E2 -14509.059} C_VEL
LIN {X 0,Y 340.048,Z 465.286,A -85,B 0,C 180,E1 -14509.863,E2 -14509.863} C_VEL
LIN {X 0,Y 340.838,Z 452.66,A -85,B 0,C 180,E1 -14510.444,E2 -14510.444} C_VEL
LIN {X 0,Y 341.351,Z 438.229,A -85,B 0,C 180,E1 -14510.839,E2 -14510.839} C_VEL
LIN {X 0,Y 342.518,Z 376.311,A -85,B 0,C 180,E1 -14512.195,E2 -14512.195} C_VEL
LIN {X 0,Y 336.888,Z 339.046,A -85,B 0,C 180,E1 -14513.423,E2 -14513.423} C_VEL
LIN {X 0,Y 337.856,Z 330.241,A -85,B 0,C 180,E1 -14515.574,E2 -14515.574} C_VEL
LIN {X 0,Y 336.606,Z 322.359,A -85,B 0,C 180,E1 -14517.666,E2 -14517.666} C_VEL
LIN {X 0,Y 333.805,Z 309.54,A -85,B 0,C 180,E1 -14521.236,E2 -14521.236} C_VEL
LIN {X 0,Y 333.696,Z 308.918,A -85,B 0,C 180,E1 -14521.423,E2 -14521.423} C_VEL
LIN {X 0,Y 333.691,Z 308.917,A -85,B 0,C 180,E1 -14524.775,E2 -14524.775} C_VEL
LIN {X 0,Y 333.657,Z 308.921,A -85,B 0,C 180,E1 -14527.652,E2 -14527.652} C_VEL
LIN {X 0,Y 333.652,Z 308.923,A -85,B 0,C 180,E1 -14530.768,E2 -14530.768} C_VEL
LIN {X 0,Y 333.597,Z 308.932,A -85,B 0,C 180,E1 -14534.251,E2 -14534.251} C_VEL
LIN {X 0,Y 333.645,Z 308.921,A -85,B 0,C 180,E1 -14537.619,E2 -14537.619} C_VEL
LIN {X 0,Y 333.656,Z 308.921,A -85,B 0,C 180,E1 -14541.203,E2 -14541.203} C_VEL
LIN {X 0,Y 333.678,Z 308.917,A -85,B 0,C 180,E1 -14543.861,E2 -14543.861} C_VEL
LIN {X 0,Y 333.646,Z 308.922,A -85,B 0,C 180,E1 -14547.414,E2 -14547.414} C_VEL
LIN {X 0,Y 333.69,Z 308.919,A -85,B 0,C 180,E1 -14551.026,E2 -14551.026} C_VEL
LIN {X 0,Y 333.735,Z 308.91,A -85,B 0,C 180,E1 -14553.754,E2 -14553.754} C_VEL
LIN {X 0,Y 333.657,Z 308.92,A -85,B 0,C 180,E1 -14557.719,E2 -14557.719} C_VEL
LIN {X 0,Y 333.74,Z 308.91,A -85,B 0,C 180,E1 -14561.586,E2 -14561.586} C_VEL
LIN {X 0,Y 333.809,Z 308.902,A -85,B 0,C 180,E1 -14565.577,E2 -14565.577} C_VEL
LIN {X 0,Y 333.815,Z 308.904,A -85,B 0,C 180,E1 -14569.077,E2 -14569.077} C_VEL
LIN {X 0,Y 334.004,Z 308.877,A -85,B 0,C 180,E1 -14572.747,E2 -14572.747} C_VEL
LIN {X 0,Y 333.799,Z 308.905,A -85,B 0,C 180,E1 -14575.169,E2 -14575.169} C_VEL
LIN {X 0,Y 334.099,Z 308.867,A -85,B 0,C 180,E1 -14577.589,E2 -14577.589} C_VEL
LIN {X 0,Y 334.184,Z 308.854,A -85,B 0,C 180,E1 -14580,E2 -14580} C_VEL
LIN {X 0,Y 334.098,Z 308.864,A -85,B 0,C 180,E1 -14582.411,E2 -14582.411} C_VEL
LIN {X 0,Y 333.957,Z 308.882,A -85,B 0,C 180,E1 -14586.506,E2 -14586.506} C_VEL
LIN {X 0,Y 333.818,Z 308.905,A -85,B 0,C 180,E1 -14589.696,E2 -14589.696} C_VEL
LIN {X 0,Y 333.791,Z 308.905,A -85,B 0,C 180,E1 -14593.392,E2 -14593.392} C_VEL
LIN {X 0,Y 333.756,Z 308.913,A -85,B 0,C 180,E1 -14595.887,E2 -14595.887} C_VEL
LIN {X 0,Y 333.723,Z 308.911,A -85,B 0,C 180,E1 -14598.617,E2 -14598.617} C_VEL
LIN {X 0,Y 333.649,Z 308.924,A -85,B 0,C 180,E1 -14602.281,E2 -14602.281} C_VEL
LIN {X 0,Y 333.655,Z 308.92,A -85,B 0,C 180,E1 -14605.077,E2 -14605.077} C_VEL
LIN {X 0,Y 333.624,Z 308.923,A -85,B 0,C 180,E1 -14608.981,E2 -14608.981} C_VEL
LIN {X 0,Y 333.639,Z 308.923,A -85,B 0,C 180,E1 -14612.585,E2 -14612.585} C_VEL
LIN {X 0,Y 333.674,Z 308.921,A -85,B 0,C 180,E1 -14616.139,E2 -14616.139} C_VEL
LIN {X 0,Y 333.604,Z 308.926,A -85,B 0,C 180,E1 -14619.199,E2 -14619.199} C_VEL
LIN {X 0,Y 333.614,Z 308.931,A -85,B 0,C 180,E1 -14622.495,E2 -14622.495} C_VEL
LIN {X 0,Y 333.587,Z 308.929,A -85,B 0,C 180,E1 -14625.952,E2 -14625.952} C_VEL
LIN {X 0,Y 333.602,Z 308.927,A -85,B 0,C 180,E1 -14629.325,E2 -14629.325} C_VEL
LIN {X 0,Y 333.652,Z 308.922,A -85,B 0,C 180,E1 -14633.171,E2 -14633.171} C_VEL
LIN {X 0,Y 333.626,Z 308.929,A -85,B 0,C 180,E1 -14636.788,E2 -14636.788} C_VEL
LIN {X 0,Y 333.656,Z 308.92,A -85,B 0,C 180,E1 -14639.724,E2 -14639.724} C_VEL
LIN {X 0,Y 333.656,Z 308.92,A -85,B 0,C 180,E1 -14643.745,E2 -14643.745} C_VEL
LIN {X 0,Y 333.66,Z 308.92,A -85,B 0,C 180,E1 -14646.407,E2 -14646.407} C_VEL
LIN {X 0,Y 333.678,Z 308.917,A -85,B 0,C 180,E1 -14650.303,E2 -14650.303} C_VEL
LIN {X 0,Y 333.725,Z 308.914,A -85,B 0,C 180,E1 -14652.85,E2 -14652.85} C_VEL
LIN {X 0,Y 333.802,Z 308.902,A -85,B 0,C 180,E1 -14656.606,E2 -14656.606} C_VEL
LIN {X 0,Y 333.824,Z 308.899,A -85,B 0,C 180,E1 -14660.301,E2 -14660.301} C_VEL
LIN {X 0,Y 333.96,Z 308.882,A -85,B 0,C 180,E1 -14662.743,E2 -14662.743} C_VEL
LIN {X 0,Y 333.78,Z 308.907,A -85,B 0,C 180,E1 -14665.165,E2 -14665.165} C_VEL
LIN {X 0,Y 334.067,Z 308.875,A -85,B 0,C 180,E1 -14667.585,E2 -14667.585} C_VEL
LIN {X 0,Y 334.06,Z 308.871,A -85,B 0,C 180,E1 -14671.201,E2 -14671.201} C_VEL
LIN {X 0,Y 334.068,Z 308.869,A -85,B 0,C 180,E1 -14672.407,E2 -14672.407} C_VEL
LIN {X 0,Y 333.954,Z 308.927,A -85,B 0,C 180,E1 -14676.491,E2 -14676.491} C_VEL
LIN {X 0,Y 335.258,Z 315.922,A -85,B 0,C 180,E1 -14678.547,E2 -14678.547} C_VEL
LIN {X 0,Y 341.024,Z 332.638,A -85,B 0,C 180,E1 -14679.317,E2 -14679.317} C_VEL
LIN {X 0,Y 343.194,Z 343.854,A -85,B 0,C 180,E1 -14679.715,E2 -14679.715} C_VEL
LIN {X 0,Y 341.331,Z 423.249,A -85,B 0,C 180,E1 -14681.463,E2 -14681.463} C_VEL
LIN {X 0,Y 340.75,Z 436.873,A -85,B 0,C 180,E1 -14682.011,E2 -14682.011} C_VEL
LIN {X 0,Y 339.952,Z 449.489,A -85,B 0,C 180,E1 -14682.76,E2 -14682.76} C_VEL
LIN {X 0,Y 338.952,Z 461.65,A -85,B 0,C 180,E1 -14683.747,E2 -14683.747} C_VEL
LIN {X 0,Y 337.846,Z 472.839,A -85,B 0,C 180,E1 -14684.913,E2 -14684.913} C_VEL
LIN {X 0,Y 336.724,Z 483.023,A -85,B 0,C 180,E1 -14686.239,E2 -14686.239} C_VEL
LIN {X 0,Y 335.742,Z 491.858,A -85,B 0,C 180,E1 -14687.664,E2 -14687.664} C_VEL
LIN {X 0,Y 334.723,Z 500.185,A -85,B 0,C 180,E1 -14689.308,E2 -14689.308} C_VEL
LIN {X 0,Y 333.909,Z 507.009,A -85,B 0,C 180,E1 -14690.96,E2 -14690.96} C_VEL
LIN {X 0,Y 333.231,Z 513.611,A -85,B 0,C 180,E1 -14692.959,E2 -14692.959} C_VEL
LIN {X 0,Y 332.685,Z 518.741,A -85,B 0,C 180,E1 -14694.986,E2 -14694.986} C_VEL
LIN {X 0,Y 332.156,Z 522.919,A -85,B 0,C 180,E1 -14697.293,E2 -14697.293} C_VEL
LIN {X 0,Y 331.873,Z 525.652,A -85,B 0,C 180,E1 -14699.744,E2 -14699.744} C_VEL
LIN {X 0,Y 331.786,Z 526.686,A -85,B 0,C 180,E1 -14702.081,E2 -14702.081} C_VEL
LIN {X 0,Y 331.895,Z 526.314,A -85,B 0,C 180,E1 -14704.326,E2 -14704.326} C_VEL
LIN {X 0,Y 332.163,Z 524.64,A -85,B 0,C 180,E1 -14706.484,E2 -14706.484} C_VEL
LIN {X 0,Y 332.58,Z 521.767,A -85,B 0,C 180,E1 -14708.567,E2 -14708.567} C_VEL
LIN {X 0,Y 333.267,Z 517.197,A -85,B 0,C 180,E1 -14710.815,E2 -14710.815} C_VEL
LIN {X 0,Y 333.895,Z 512.5,A -85,B 0,C 180,E1 -14712.549,E2 -14712.549} C_VEL
LIN {X 0,Y 334.132,Z 510.943,A -85,B 0,C 180,E1 -14713.04,E2 -14713.04} C_VEL
LIN {X 0,Y 333.951,Z 508.088,A -85,B 0,C 180,E1 -14713.927,E2 -14713.927} C_VEL
LIN {X 0,Y 331.984,Z 503.125,A -85,B 0,C 180,E1 -14715.366,E2 -14715.366} C_VEL
LIN {X 0,Y 330.105,Z 497.578,A -85,B 0,C 180,E1 -14716.751,E2 -14716.751} C_VEL
LIN {X 0,Y 330.057,Z 493.764,A -85,B 0,C 180,E1 -14717.536,E2 -14717.536} C_VEL
LIN {X 0,Y 331.534,Z 484.171,A -85,B 0,C 180,E1 -14719.15,E2 -14719.15} C_VEL
LIN {X 0,Y 332.665,Z 474.981,A -85,B 0,C 180,E1 -14720.41,E2 -14720.41} C_VEL
LIN {X 0,Y 334.212,Z 463.237,A -85,B 0,C 180,E1 -14721.675,E2 -14721.675} C_VEL
LIN {X 0,Y 335.359,Z 451.718,A -85,B 0,C 180,E1 -14722.65,E2 -14722.65} C_VEL
LIN {X 0,Y 336.333,Z 438.98,A -85,B 0,C 180,E1 -14723.455,E2 -14723.455} C_VEL
LIN {X 0,Y 337.023,Z 426.592,A -85,B 0,C 180,E1 -14723.99,E2 -14723.99} C_VEL
LIN {X 0,Y 337.694,Z 404.666,A -85,B 0,C 180,E1 -14724.537,E2 -14724.537} C_VEL
LIN {X 0,Y 339.282,Z 345.316,A -85,B 0,C 180,E1 -14725.876,E2 -14725.876} C_VEL
LIN {X 0,Y 337.748,Z 338.406,A -85,B 0,C 180,E1 -14726.183,E2 -14726.183} C_VEL
LIN {X 0,Y 331.905,Z 324.309,A -85,B 0,C 180,E1 -14727.075,E2 -14727.075} C_VEL
LIN {X 0,Y 328.178,Z 316.224,A -85,B 0,C 180,E1 -14727.675,E2 -14727.675} C_VEL
LIN {X 0,Y 326.644,Z 309.799,A -85,B 0,C 180,E1 -14729.662,E2 -14729.662} C_VEL
LIN {X 0,Y 326.645,Z 309.802,A -85,B 0,C 180,E1 -14733.139,E2 -14733.139} C_VEL
LIN {X 0,Y 326.61,Z 309.81,A -85,B 0,C 180,E1 -14735.868,E2 -14735.868} C_VEL
LIN {X 0,Y 326.615,Z 309.805,A -85,B 0,C 180,E1 -14739.862,E2 -14739.862} C_VEL
LIN {X 0,Y 326.655,Z 309.8,A -85,B 0,C 180,E1 -14742.47,E2 -14742.47} C_VEL
LIN {X 0,Y 326.712,Z 309.786,A -85,B 0,C 180,E1 -14746.313,E2 -14746.313} C_VEL
LIN {X 0,Y 326.739,Z 309.78,A -85,B 0,C 180,E1 -14750.091,E2 -14750.091} C_VEL
LIN {X 0,Y 326.909,Z 309.759,A -85,B 0,C 180,E1 -14752.589,E2 -14752.589} C_VEL
LIN {X 0,Y 326.73,Z 309.782,A -85,B 0,C 180,E1 -14755.064,E2 -14755.064} C_VEL
LIN {X 0,Y 327.001,Z 309.75,A -85,B 0,C 180,E1 -14757.536,E2 -14757.536} C_VEL
LIN {X 0,Y 327.133,Z 309.725,A -85,B 0,C 180,E1 -14760,E2 -14760} C_VEL
LIN {X 0,Y 327.002,Z 309.752,A -85,B 0,C 180,E1 -14762.464,E2 -14762.464} C_VEL
LIN {X 0,Y 326.944,Z 309.758,A -85,B 0,C 180,E1 -14766.17,E2 -14766.17} C_VEL
LIN {X 0,Y 326.769,Z 309.78,A -85,B 0,C 180,E1 -14769.908,E2 -14769.908} C_VEL
LIN {X 0,Y 326.716,Z 309.786,A -85,B 0,C 180,E1 -14773.687,E2 -14773.687} C_VEL
LIN {X 0,Y 326.657,Z 309.791,A -85,B 0,C 180,E1 -14777.53,E2 -14777.53} C_VEL
LIN {X 0,Y 326.644,Z 309.785,A -85,B 0,C 180,E1 -14780.136,E2 -14780.136} C_VEL
LIN {X 0,Y 326.63,Z 309.787,A -85,B 0,C 180,E1 -14784.131,E2 -14784.131} C_VEL
LIN {X 0,Y 326.646,Z 309.794,A -85,B 0,C 180,E1 -14786.861,E2 -14786.861} C_VEL
LIN {X 0,Y 326.602,Z 309.799,A -85,B 0,C 180,E1 -14790.615,E2 -14790.615} C_VEL
LIN {X 0,Y 326.574,Z 309.804,A -85,B 0,C 180,E1 -14794.023,E2 -14794.023} C_VEL
LIN {X 0,Y 326.646,Z 309.799,A -85,B 0,C 180,E1 -14797.255,E2 -14797.255} C_VEL
LIN {X 0,Y 326.616,Z 309.801,A -85,B 0,C 180,E1 -14800.205,E2 -14800.205} C_VEL
LIN {X 0,Y 326.629,Z 309.802,A -85,B 0,C 180,E1 -14803.514,E2 -14803.514} C_VEL
LIN {X 0,Y 326.624,Z 309.804,A -85,B 0,C 180,E1 -14807.019,E2 -14807.019} C_VEL
LIN {X 0,Y 326.622,Z 309.801,A -85,B 0,C 180,E1 -14810.771,E2 -14810.771} C_VEL
LIN {X 0,Y 326.592,Z 309.801,A -85,B 0,C 180,E1 -14814.486,E2 -14814.486} C_VEL
LIN {X 0,Y 326.595,Z 309.94,A -85,B 0,C 180,E1 -14817.06,E2 -14817.06} C_VEL
LIN {X 0,Y 328.944,Z 319.327,A -85,B 0,C 180,E1 -14819.869,E2 -14819.869} C_VEL
LIN {X 0,Y 330.918,Z 328.407,A -85,B 0,C 180,E1 -14822.438,E2 -14822.438} C_VEL
LIN {X 0,Y 331.776,Z 333.955,A -85,B 0,C 180,E1 -14823.931,E2 -14823.931} C_VEL
LIN {X 0,Y 331.405,Z 337.124,A -85,B 0,C 180,E1 -14824.701,E2 -14824.701} C_VEL
LIN {X 0,Y 335.966,Z 360.809,A -85,B 0,C 180,E1 -14825.727,E2 -14825.727} C_VEL
LIN {X 0,Y 338.525,Z 378.939,A -85,B 0,C 180,E1 -14826.399,E2 -14826.399} C_VEL
LIN {X 0,Y 336.691,Z 446.299,A -85,B 0,C 180,E1 -14827.937,E2 -14827.937} C_VEL
LIN {X 0,Y 335.847,Z 459.292,A -85,B 0,C 180,E1 -14828.443,E2 -14828.443} C_VEL
LIN {X 0,Y 334.726,Z 471.929,A -85,B 0,C 180,E1 -14829.174,E2 -14829.174} C_VEL
LIN {X 0,Y 333.408,Z 484.056,A -85,B 0,C 180,E1 -14830.135,E2 -14830.135} C_VEL
LIN {X 0,Y 331.867,Z 495.611,A -85,B 0,C 180,E1 -14831.324,E2 -14831.324} C_VEL
LIN {X 0,Y 330.44,Z 506.051,A -85,B 0,C 180,E1 -14832.682,E2 -14832.682} C_VEL
LIN {X 0,Y 329.129,Z 515.474,A -85,B 0,C 180,E1 -14834.207,E2 -14834.207} C_VEL
LIN {X 0,Y 327.755,Z 524.6,A -85,B 0,C 180,E1 -14836.046,E2 -14836.046} C_VEL
LIN {X 0,Y 326.574,Z 531.977,A -85,B 0,C 180,E1 -14837.893,E2 -14837.893} C_VEL
LIN {X 0,Y 325.747,Z 538.755,A -85,B 0,C 180,E1 -14840.066,E2 -14840.066} C_VEL
LIN {X 0,Y 325.258,Z 543.25,A -85,B 0,C 180,E1 -14841.931,E2 -14841.931} C_VEL
LIN {X 0,Y 324.945,Z 547.285,A -85,B 0,C 180,E1 -14844.214,E2 -14844.214} C_VEL
LIN {X 0,Y 324.9,Z 549.685,A -85,B 0,C 180,E1 -14846.284,E2 -14846.284} C_VEL
LIN {X 0,Y 324.858,Z 550.582,A -85,B 0,C 180,E1 -14847.524,E2 -14847.524} C_VEL
LIN {X 0,Y 324.879,Z 551.037,A -85,B 0,C 180,E1 -14848.765,E2 -14848.765} C_VEL
LIN {X 0,Y 324.948,Z 551.097,A -85,B 0,C 180,E1 -14850.004,E2 -14850.004} C_VEL
LIN {X 0,Y 324.894,Z 550.76,A -85,B 0,C 180,E1 -14851.243,E2 -14851.243} C_VEL
LIN {X 0,Y 324.862,Z 550.02,A -85,B 0,C 180,E1 -14852.484,E2 -14852.484} C_VEL
LIN {X 0,Y 324.928,Z 548.829,A -85,B 0,C 180,E1 -14853.724,E2 -14853.724} C_VEL
LIN {X 0,Y 324.913,Z 546.014,A -85,B 0,C 180,E1 -14855.73,E2 -14855.73} C_VEL
LIN {X 0,Y 325.232,Z 541.21,A -85,B 0,C 180,E1 -14858.078,E2 -14858.078} C_VEL
LIN {X 0,Y 325.728,Z 535.075,A -85,B 0,C 180,E1 -14860.257,E2 -14860.257} C_VEL
LIN {X 0,Y 326.443,Z 528.345,A -85,B 0,C 180,E1 -14862.12,E2 -14862.12} C_VEL
LIN {X 0,Y 327.479,Z 519.988,A -85,B 0,C 180,E1 -14863.974,E2 -14863.974} C_VEL
LIN {X 0,Y 328.582,Z 511.026,A -85,B 0,C 180,E1 -14865.57,E2 -14865.57} C_VEL
LIN {X 0,Y 329.673,Z 500.764,A -85,B 0,C 180,E1 -14867.048,E2 -14867.048} C_VEL
LIN {X 0,Y 330.915,Z 490.255,A -85,B 0,C 180,E1 -14868.259,E2 -14868.259} C_VEL
LIN {X 0,Y 332.134,Z 478.695,A -85,B 0,C 180,E1 -14869.31,E2 -14869.31} C_VEL
LIN {X 0,Y 333.18,Z 466.732,A -85,B 0,C 180,E1 -14870.129,E2 -14870.129} C_VEL
LIN {X 0,Y 334.051,Z 452.979,A -85,B 0,C 180,E1 -14870.798,E2 -14870.798} C_VEL
LIN {X 0,Y 334.586,Z 439.753,A -85,B 0,C 180,E1 -14871.184,E2 -14871.184} C_VEL
LIN {X 0,Y 335.858,Z 377.188,A -85,B 0,C 180,E1 -14872.581,E2 -14872.581} C_VEL
LIN {X 0,Y 330.326,Z 340.628,A -85,B 0,C 180,E1 -14873.813,E2 -14873.813} C_VEL
LIN {X 0,Y 330.067,Z 338.683,A -85,B 0,C 180,E1 -14873.908,E2 -14873.908} C_VEL
LIN {X 0,Y 330.906,Z 331.054,A -85,B 0,C 180,E1 -14875.813,E2 -14875.813} C_VEL
LIN {X 0,Y 329.522,Z 323.072,A -85,B 0,C 180,E1 -14877.986,E2 -14877.986} C_VEL
LIN {X 0,Y 326.661,Z 309.796,A -85,B 0,C 180,E1 -14881.79,E2 -14881.79} C_VEL
LIN {X 0,Y 326.618,Z 309.798,A -85,B 0,C 180,E1 -14885.521,E2 -14885.521} C_VEL
LIN {X 0,Y 326.617,Z 309.796,A -85,B 0,C 180,E1 -14889.228,E2 -14889.228} C_VEL
LIN {X 0,Y 326.581,Z 309.802,A -85,B 0,C 180,E1 -14892.973,E2 -14892.973} C_VEL
LIN {X 0,Y 326.58,Z 309.803,A -85,B 0,C 180,E1 -14897.029,E2 -14897.029} C_VEL
LIN {X 0,Y 326.615,Z 309.801,A -85,B 0,C 180,E1 -14900.774,E2 -14900.774} C_VEL
LIN {X 0,Y 326.615,Z 309.802,A -85,B 0,C 180,E1 -14904.481,E2 -14904.481} C_VEL
LIN {X 0,Y 326.61,Z 309.798,A -85,B 0,C 180,E1 -14907.456,E2 -14907.456} C_VEL
LIN {X 0,Y 326.635,Z 309.796,A -85,B 0,C 180,E1 -14910.338,E2 -14910.338} C_VEL
LIN {X 0,Y 326.684,Z 309.791,A -85,B 0,C 180,E1 -14913.142,E2 -14913.142} C_VEL
LIN {X 0,Y 326.65,Z 309.792,A -85,B 0,C 180,E1 -14915.871,E2 -14915.871} C_VEL
LIN {X 0,Y 326.617,Z 309.796,A -85,B 0,C 180,E1 -14919.862,E2 -14919.862} C_VEL
LIN {X 0,Y 326.707,Z 309.783,A -85,B 0,C 180,E1 -14923.761,E2 -14923.761} C_VEL
LIN {X 0,Y 326.756,Z 309.778,A -85,B 0,C 180,E1 -14926.314,E2 -14926.314} C_VEL
LIN {X 0,Y 326.783,Z 309.776,A -85,B 0,C 180,E1 -14930.093,E2 -14930.093} C_VEL
LIN {X 0,Y 326.954,Z 309.755,A -85,B 0,C 180,E1 -14932.59,E2 -14932.59} C_VEL
LIN {X 0,Y 326.985,Z 309.751,A -85,B 0,C 180,E1 -14933.831,E2 -14933.831} C_VEL
LIN {X 0,Y 327.039,Z 309.745,A -85,B 0,C 180,E1 -14937.537,E2 -14937.537} C_VEL
LIN {X 0,Y 327.138,Z 309.731,A -85,B 0,C 180,E1 -14940,E2 -14940} C_VEL
LIN {X 0,Y 327.039,Z 309.743,A -85,B 0,C 180,E1 -14942.463,E2 -14942.463} C_VEL
LIN {X 0,Y 326.918,Z 309.759,A -85,B 0,C 180,E1 -14946.495,E2 -14946.495} C_VEL
LIN {X 0,Y 326.781,Z 309.779,A -85,B 0,C 180,E1 -14949.907,E2 -14949.907} C_VEL
LIN {X 0,Y 326.756,Z 309.784,A -85,B 0,C 180,E1 -14953.686,E2 -14953.686} C_VEL
LIN {X 0,Y 326.662,Z 309.793,A -85,B 0,C 180,E1 -14957.53,E2 -14957.53} C_VEL
LIN {X 0,Y 326.614,Z 309.798,A -85,B 0,C 180,E1 -14961.457,E2 -14961.457} C_VEL
LIN {X 0,Y 326.584,Z 309.801,A -85,B 0,C 180,E1 -14965.493,E2 -14965.493} C_VEL
LIN {X 0,Y 326.589,Z 309.803,A -85,B 0,C 180,E1 -14968.257,E2 -14968.257} C_VEL
LIN {X 0,Y 326.567,Z 309.798,A -85,B 0,C 180,E1 -14971.098,E2 -14971.098} C_VEL
LIN {X 0,Y 326.607,Z 309.799,A -85,B 0,C 180,E1 -14974.02,E2 -14974.02} C_VEL
LIN {X 0,Y 326.623,Z 309.796,A -85,B 0,C 180,E1 -14977.236,E2 -14977.236} C_VEL
LIN {X 0,Y 326.538,Z 309.807,A -85,B 0,C 180,E1 -14981.122,E2 -14981.122} C_VEL
LIN {X 0,Y 326.521,Z 309.813,A -85,B 0,C 180,E1 -14984.74,E2 -14984.74} C_VEL
LIN {X 0,Y 326.55,Z 309.806,A -85,B 0,C 180,E1 -14988.148,E2 -14988.148} C_VEL
LIN {X 0,Y 326.566,Z 309.804,A -85,B 0,C 180,E1 -14991.381,E2 -14991.381} C_VEL
LIN {X 0,Y 326.595,Z 309.805,A -85,B 0,C 180,E1 -14994.858,E2 -14994.858} C_VEL
LIN {X 0,Y 326.601,Z 309.8,A -85,B 0,C 180,E1 -14997.453,E2 -14997.453} C_VEL
LIN {X 0,Y 326.589,Z 309.801,A -85,B 0,C 180,E1 -15000.331,E2 -15000.331} C_VEL
LIN {X 0,Y 326.639,Z 309.796,A -85,B 0,C 180,E1 -15004.509,E2 -15004.509} C_VEL
LIN {X 0,Y 326.621,Z 309.798,A -85,B 0,C 180,E1 -15008.541,E2 -15008.541} C_VEL
LIN {X 0,Y 326.67,Z 309.791,A -85,B 0,C 180,E1 -15012.468,E2 -15012.468} C_VEL
LIN {X 0,Y 326.765,Z 309.778,A -85,B 0,C 180,E1 -15016.312,E2 -15016.312} C_VEL
LIN {X 0,Y 326.787,Z 309.776,A -85,B 0,C 180,E1 -15020.09,E2 -15020.09} C_VEL
LIN {X 0,Y 326.944,Z 309.759,A -85,B 0,C 180,E1 -15023.826,E2 -15023.826} C_VEL
LIN {X 0,Y 327.011,Z 309.754,A -85,B 0,C 180,E1 -15027.533,E2 -15027.533} C_VEL
LIN {X 0,Y 327.03,Z 309.747,A -85,B 0,C 180,E1 -15031.227,E2 -15031.227} C_VEL
LIN {X 0,Y 326.756,Z 309.786,A -85,B 0,C 180,E1 -15033.695,E2 -15033.695} C_VEL
LIN {X 0,Y 326.945,Z 309.852,A -85,B 0,C 180,E1 -15036.166,E2 -15036.166} C_VEL
LIN {X 0,Y 328.044,Z 315.923,A -85,B 0,C 180,E1 -15038.039,E2 -15038.039} C_VEL
LIN {X 0,Y 334.503,Z 334.2,A -85,B 0,C 180,E1 -15038.933,E2 -15038.933} C_VEL
LIN {X 0,Y 336.5,Z 345.139,A -85,B 0,C 180,E1 -15039.322,E2 -15039.322} C_VEL
LIN {X 0,Y 334.606,Z 423.468,A -85,B 0,C 180,E1 -15041.083,E2 -15041.083} C_VEL
LIN {X 0,Y 334.003,Z 437.101,A -85,B 0,C 180,E1 -15041.641,E2 -15041.641} C_VEL
LIN {X 0,Y 333.171,Z 449.733,A -85,B 0,C 180,E1 -15042.405,E2 -15042.405} C_VEL
LIN {X 0,Y 332.254,Z 461.129,A -85,B 0,C 180,E1 -15043.34,E2 -15043.34} C_VEL
LIN {X 0,Y 330.985,Z 473.095,A -85,B 0,C 180,E1 -15044.6,E2 -15044.6} C_VEL
LIN {X 0,Y 329.713,Z 484.124,A -85,B 0,C 180,E1 -15046.082,E2 -15046.082} C_VEL
LIN {X 0,Y 328.597,Z 493.891,A -85,B 0,C 180,E1 -15047.739,E2 -15047.739} C_VEL
LIN {X 0,Y 327.638,Z 501.381,A -85,B 0,C 180,E1 -15049.296,E2 -15049.296} C_VEL
LIN {X 0,Y 326.77,Z 508.503,A -85,B 0,C 180,E1 -15051.11,E2 -15051.11} C_VEL
LIN {X 0,Y 326.185,Z 513.876,A -85,B 0,C 180,E1 -15052.813,E2 -15052.813} C_VEL
LIN {X 0,Y 325.607,Z 519.177,A -85,B 0,C 180,E1 -15054.968,E2 -15054.968} C_VEL
LIN {X 0,Y 325.128,Z 522.819,A -85,B 0,C 180,E1 -15056.99,E2 -15056.99} C_VEL
LIN {X 0,Y 324.891,Z 524.685,A -85,B 0,C 180,E1 -15058.411,E2 -15058.411} C_VEL
LIN {X 0,Y 324.745,Z 526.118,A -85,B 0,C 180,E1 -15060.041,E2 -15060.041} C_VEL
LIN {X 0,Y 324.692,Z 526.997,A -85,B 0,C 180,E1 -15062.418,E2 -15062.418} C_VEL
LIN {X 0,Y 324.837,Z 526.437,A -85,B 0,C 180,E1 -15064.699,E2 -15064.699} C_VEL
LIN {X 0,Y 325.14,Z 524.61,A -85,B 0,C 180,E1 -15066.892,E2 -15066.892} C_VEL
LIN {X 0,Y 325.597,Z 521.622,A -85,B 0,C 180,E1 -15069.008,E2 -15069.008} C_VEL
LIN {X 0,Y 326.279,Z 517.442,A -85,B 0,C 180,E1 -15071.071,E2 -15071.071} C_VEL
LIN {X 0,Y 327.134,Z 511.617,A -85,B 0,C 180,E1 -15073.21,E2 -15073.21} C_VEL
LIN {X 0,Y 328.179,Z 505.232,A -85,B 0,C 180,E1 -15075.033,E2 -15075.033} C_VEL
LIN {X 0,Y 329.577,Z 496.698,A -85,B 0,C 180,E1 -15076.97,E2 -15076.97} C_VEL
LIN {X 0,Y 330.057,Z 493.764,A -85,B 0,C 180,E1 -15077.536,E2 -15077.536} C_VEL
LIN {X 0,Y 330.022,Z 489.787,A -85,B 0,C 180,E1 -15078.296,E2 -15078.296} C_VEL
LIN {X 0,Y 328.263,Z 483.14,A -85,B 0,C 180,E1 -15079.543,E2 -15079.543} C_VEL
LIN {X 0,Y 326.584,Z 476.038,A -85,B 0,C 180,E1 -15080.708,E2 -15080.708} C_VEL
LIN {X 0,Y 326.653,Z 471.299,A -85,B 0,C 180,E1 -15081.326,E2 -15081.326} C_VEL
LIN {X 0,Y 327.954,Z 460.443,A -85,B 0,C 180,E1 -15082.446,E2 -15082.446} C_VEL
LIN {X 0,Y 329.208,Z 448.384,A -85,B 0,C 180,E1 -15083.398,E2 -15083.398} C_VEL
LIN {X 0,Y 330.156,Z 435.424,A -85,B 0,C 180,E1 -15084.155,E2 -15084.155} C_VEL
LIN {X 0,Y 330.808,Z 423.154,A -85,B 0,C 180,E1 -15084.625,E2 -15084.625} C_VEL
LIN {X 0,Y 332.871,Z 346.03,A -85,B 0,C 180,E1 -15086.424,E2 -15086.424} C_VEL
LIN {X 0,Y 331.585,Z 340.617,A -85,B 0,C 180,E1 -15086.681,E2 -15086.681} C_VEL
LIN {X 0,Y 325.665,Z 326.402,A -85,B 0,C 180,E1 -15087.625,E2 -15087.625} C_VEL
LIN {X 0,Y 321.03,Z 316.638,A -85,B 0,C 180,E1 -15088.363,E2 -15088.363} C_VEL
LIN {X 0,Y 319.579,Z 310.68,A -85,B 0,C 180,E1 -15090.252,E2 -15090.252} C_VEL
LIN {X 0,Y 319.596,Z 310.682,A -85,B 0,C 180,E1 -15094.352,E2 -15094.352} C_VEL
LIN {X 0,Y 319.529,Z 310.692,A -85,B 0,C 180,E1 -15098.043,E2 -15098.043} C_VEL
LIN {X 0,Y 319.648,Z 310.669,A -85,B 0,C 180,E1 -15100.96,E2 -15100.96} C_VEL
LIN {X 0,Y 319.688,Z 310.664,A -85,B 0,C 180,E1 -15105.275,E2 -15105.275} C_VEL
LIN {X 0,Y 319.691,Z 310.657,A -85,B 0,C 180,E1 -15109.871,E2 -15109.871} C_VEL
LIN {X 0,Y 319.896,Z 310.635,A -85,B 0,C 180,E1 -15113.693,E2 -15113.693} C_VEL
LIN {X 0,Y 319.945,Z 310.63,A -85,B 0,C 180,E1 -15117.482,E2 -15117.482} C_VEL
LIN {X 0,Y 320.085,Z 310.603,A -85,B 0,C 180,E1 -15120,E2 -15120} C_VEL
LIN {X 0,Y 319.946,Z 310.63,A -85,B 0,C 180,E1 -15122.518,E2 -15122.518} C_VEL
LIN {X 0,Y 319.899,Z 310.636,A -85,B 0,C 180,E1 -15126.306,E2 -15126.306} C_VEL
LIN {X 0,Y 319.796,Z 310.644,A -85,B 0,C 180,E1 -15128.849,E2 -15128.849} C_VEL
LIN {X 0,Y 319.639,Z 310.66,A -85,B 0,C 180,E1 -15132.702,E2 -15132.702} C_VEL
LIN {X 0,Y 319.642,Z 310.663,A -85,B 0,C 180,E1 -15135.298,E2 -15135.298} C_VEL
LIN {X 0,Y 319.639,Z 310.664,A -85,B 0,C 180,E1 -15139.257,E2 -15139.257} C_VEL
LIN {X 0,Y 319.578,Z 310.671,A -85,B 0,C 180,E1 -15143.319,E2 -15143.319} C_VEL
LIN {X 0,Y 319.598,Z 310.671,A -85,B 0,C 180,E1 -15146.091,E2 -15146.091} C_VEL
LIN {X 0,Y 319.551,Z 310.672,A -85,B 0,C 180,E1 -15148.937,E2 -15148.937} C_VEL
LIN {X 0,Y 319.496,Z 310.681,A -85,B 0,C 180,E1 -15151.866,E2 -15151.866} C_VEL
LIN {X 0,Y 319.564,Z 310.675,A -85,B 0,C 180,E1 -15155.552,E2 -15155.552} C_VEL
LIN {X 0,Y 319.6,Z 310.671,A -85,B 0,C 180,E1 -15158.004,E2 -15158.004} C_VEL
LIN {X 0,Y 319.573,Z 310.678,A -85,B 0,C 180,E1 -15161.617,E2 -15161.617} C_VEL
LIN {X 0,Y 319.618,Z 310.679,A -85,B 0,C 180,E1 -15165.29,E2 -15165.29} C_VEL
LIN {X 0,Y 319.558,Z 310.683,A -85,B 0,C 180,E1 -15168.725,E2 -15168.725} C_VEL
LIN {X 0,Y 319.577,Z 310.679,A -85,B 0,C 180,E1 -15172.345,E2 -15172.345} C_VEL
LIN {X 0,Y 319.543,Z 310.682,A -85,B 0,C 180,E1 -15176.378,E2 -15176.378} C_VEL
LIN {X 0,Y 322.353,Z 322.051,A -85,B 0,C 180,E1 -15179.911,E2 -15179.911} C_VEL
LIN {X 0,Y 324.368,Z 331.611,A -85,B 0,C 180,E1 -15182.665,E2 -15182.665} C_VEL
LIN {X 0,Y 324.928,Z 335.322,A -85,B 0,C 180,E1 -15183.685,E2 -15183.685} C_VEL
LIN {X 0,Y 324.78,Z 336.819,A -85,B 0,C 180,E1 -15184.06,E2 -15184.06} C_VEL
LIN {X 0,Y 329.589,Z 361.314,A -85,B 0,C 180,E1 -15185.172,E2 -15185.172} C_VEL
LIN {X 0,Y 332.157,Z 379.499,A -85,B 0,C 180,E1 -15185.867,E2 -15185.867} C_VEL
LIN {X 0,Y 330.253,Z 446.158,A -85,B 0,C 180,E1 -15187.42,E2 -15187.42} C_VEL
LIN {X 0,Y 329.342,Z 459.461,A -85,B 0,C 180,E1 -15187.954,E2 -15187.954} C_VEL
LIN {X 0,Y 328.136,Z 472.505,A -85,B 0,C 180,E1 -15188.736,E2 -15188.736} C_VEL
LIN {X 0,Y 326.744,Z 484.364,A -85,B 0,C 180,E1 -15189.712,E2 -15189.712} C_VEL
LIN {X 0,Y 325.145,Z 495.793,A -85,B 0,C 180,E1 -15190.923,E2 -15190.923} C_VEL
LIN {X 0,Y 323.671,Z 506.139,A -85,B 0,C 180,E1 -15192.308,E2 -15192.308} C_VEL
LIN {X 0,Y 322.349,Z 515.043,A -85,B 0,C 180,E1 -15193.78,E2 -15193.78} C_VEL
LIN {X 0,Y 321.09,Z 523.191,A -85,B 0,C 180,E1 -15195.426,E2 -15195.426} C_VEL
LIN {X 0,Y 319.785,Z 530.767,A -85,B 0,C 180,E1 -15197.309,E2 -15197.309} C_VEL
LIN {X 0,Y 318.925,Z 536.876,A -85,B 0,C 180,E1 -15199.209,E2 -15199.209} C_VEL
LIN {X 0,Y 318.353,Z 541.727,A -85,B 0,C 180,E1 -15201.115,E2 -15201.115} C_VEL
LIN {X 0,Y 317.986,Z 545.459,A -85,B 0,C 180,E1 -15203.023,E2 -15203.023} C_VEL
LIN {X 0,Y 317.808,Z 548.172,A -85,B 0,C 180,E1 -15204.93,E2 -15204.93} C_VEL
LIN {X 0,Y 317.807,Z 549.465,A -85,B 0,C 180,E1 -15206.2,E2 -15206.2} C_VEL
LIN {X 0,Y 317.778,Z 550.339,A -85,B 0,C 180,E1 -15207.469,E2 -15207.469} C_VEL
LIN {X 0,Y 317.787,Z 550.777,A -85,B 0,C 180,E1 -15208.737,E2 -15208.737} C_VEL
LIN {X 0,Y 317.852,Z 550.825,A -85,B 0,C 180,E1 -15210.004,E2 -15210.004} C_VEL
LIN {X 0,Y 317.801,Z 550.475,A -85,B 0,C 180,E1 -15211.271,E2 -15211.271} C_VEL
LIN {X 0,Y 317.783,Z 549.714,A -85,B 0,C 180,E1 -15212.539,E2 -15212.539} C_VEL
LIN {X 0,Y 317.833,Z 548.505,A -85,B 0,C 180,E1 -15213.807,E2 -15213.807} C_VEL
LIN {X 0,Y 317.814,Z 545.987,A -85,B 0,C 180,E1 -15215.666,E2 -15215.666} C_VEL
LIN {X 0,Y 318.064,Z 542.269,A -85,B 0,C 180,E1 -15217.622,E2 -15217.622} C_VEL
LIN {X 0,Y 318.437,Z 537.493,A -85,B 0,C 180,E1 -15219.531,E2 -15219.531} C_VEL
LIN {X 0,Y 319.186,Z 530.305,A -85,B 0,C 180,E1 -15221.755,E2 -15221.755} C_VEL
LIN {X 0,Y 320.21,Z 522.467,A -85,B 0,C 180,E1 -15223.65,E2 -15223.65} C_VEL
LIN {X 0,Y 321.415,Z 512.891,A -85,B 0,C 180,E1 -15225.494,E2 -15225.494} C_VEL
LIN {X 0,Y 322.581,Z 502.427,A -85,B 0,C 180,E1 -15227.108,E2 -15227.108} C_VEL
LIN {X 0,Y 323.973,Z 490.884,A -85,B 0,C 180,E1 -15228.5,E2 -15228.5} C_VEL
LIN {X 0,Y 325.241,Z 479.564,A -85,B 0,C 180,E1 -15229.571,E2 -15229.571} C_VEL
LIN {X 0,Y 326.304,Z 468.06,A -85,B 0,C 180,E1 -15230.408,E2 -15230.408} C_VEL
LIN {X 0,Y 327.191,Z 454.941,A -85,B 0,C 180,E1 -15231.09,E2 -15231.09} C_VEL
LIN {X 0,Y 327.812,Z 441.885,A -85,B 0,C 180,E1 -15231.519,E2 -15231.519} C_VEL
LIN {X 0,Y 329.195,Z 378.047,A -85,B 0,C 180,E1 -15232.975,E2 -15232.975} C_VEL
LIN {X 0,Y 323.844,Z 342.419,A -85,B 0,C 180,E1 -15234.204,E2 -15234.204} C_VEL
LIN {X 0,Y 323.251,Z 338.478,A -85,B 0,C 180,E1 -15234.365,E2 -15234.365} C_VEL
LIN {X 0,Y 323.915,Z 331.841,A -85,B 0,C 180,E1 -15236.066,E2 -15236.066} C_VEL
LIN {X 0,Y 322.463,Z 323.859,A -85,B 0,C 180,E1 -15238.299,E2 -15238.299} C_VEL
LIN {X 0,Y 319.687,Z 311.09,A -85,B 0,C 180,E1 -15242.032,E2 -15242.032} C_VEL
LIN {X 0,Y 319.589,Z 310.678,A -85,B 0,C 180,E1 -15242.229,E2 -15242.229} C_VEL
LIN {X 0,Y 319.564,Z 310.679,A -85,B 0,C 180,E1 -15246.429,E2 -15246.429} C_VEL
LIN {X 0,Y 319.565,Z 310.676,A -85,B 0,C 180,E1 -15249.67,E2 -15249.67} C_VEL
LIN {X 0,Y 319.526,Z 310.68,A -85,B 0,C 180,E1 -15253.461,E2 -15253.461} C_VEL
LIN {X 0,Y 319.558,Z 310.678,A -85,B 0,C 180,E1 -15257.017,E2 -15257.017} C_VEL
LIN {X 0,Y 319.551,Z 310.681,A -85,B 0,C 180,E1 -15260.371,E2 -15260.371} C_VEL
LIN {X 0,Y 319.583,Z 310.677,A -85,B 0,C 180,E1 -15264.458,E2 -15264.458} C_VEL
LIN {X 0,Y 319.527,Z 310.681,A -85,B 0,C 180,E1 -15268.138,E2 -15268.138} C_VEL
LIN {X 0,Y 319.612,Z 310.67,A -85,B 0,C 180,E1 -15271.591,E2 -15271.591} C_VEL
LIN {X 0,Y 319.604,Z 310.672,A -85,B 0,C 180,E1 -15275.304,E2 -15275.304} C_VEL
LIN {X 0,Y 319.578,Z 310.675,A -85,B 0,C 180,E1 -15279.399,E2 -15279.399} C_VEL
LIN {X 0,Y 319.65,Z 310.663,A -85,B 0,C 180,E1 -15283.392,E2 -15283.392} C_VEL
LIN {X 0,Y 319.73,Z 310.653,A -85,B 0,C 180,E1 -15286.008,E2 -15286.008} C_VEL
LIN {X 0,Y 319.735,Z 310.655,A -85,B 0,C 180,E1 -15289.872,E2 -15289.872} C_VEL
LIN {X 0,Y 319.939,Z 310.629,A -85,B 0,C 180,E1 -15293.694,E2 -15293.694} C_VEL
LIN {X 0,Y 319.983,Z 310.622,A -85,B 0,C 180,E1 -15297.482,E2 -15297.482} C_VEL
LIN {X 0,Y 320.093,Z 310.608,A -85,B 0,C 180,E1 -15300,E2 -15300} C_VEL
LIN {X 0,Y 319.983,Z 310.622,A -85,B 0,C 180,E1 -15302.518,E2 -15302.518} C_VEL
LIN {X 0,Y 319.883,Z 310.636,A -85,B 0,C 180,E1 -15306.477,E2 -15306.477} C_VEL
LIN {X 0,Y 319.734,Z 310.655,A -85,B 0,C 180,E1 -15310.128,E2 -15310.128} C_VEL
LIN {X 0,Y 319.73,Z 310.659,A -85,B 0,C 180,E1 -15313.992,E2 -15313.992} C_VEL
LIN {X 0,Y 319.614,Z 310.673,A -85,B 0,C 180,E1 -15317.93,E2 -15317.93} C_VEL
LIN {X 0,Y 319.565,Z 310.68,A -85,B 0,C 180,E1 -15321.955,E2 -15321.955} C_VEL
LIN {X 0,Y 319.543,Z 310.683,A -85,B 0,C 180,E1 -15326.096,E2 -15326.096} C_VEL
LIN {X 0,Y 319.523,Z 310.677,A -85,B 0,C 180,E1 -15328.94,E2 -15328.94} C_VEL
LIN {X 0,Y 319.52,Z 310.677,A -85,B 0,C 180,E1 -15331.863,E2 -15331.863} C_VEL
LIN {X 0,Y 319.58,Z 310.672,A -85,B 0,C 180,E1 -15335.541,E2 -15335.541} C_VEL
LIN {X 0,Y 319.519,Z 310.681,A -85,B 0,C 180,E1 -15339.634,E2 -15339.634} C_VEL
LIN {X 0,Y 319.492,Z 310.683,A -85,B 0,C 180,E1 -15343.453,E2 -15343.453} C_VEL
LIN {X 0,Y 319.492,Z 310.686,A -85,B 0,C 180,E1 -15347.004,E2 -15347.004} C_VEL
LIN {X 0,Y 319.52,Z 310.683,A -85,B 0,C 180,E1 -15350.365,E2 -15350.365} C_VEL
LIN {X 0,Y 319.546,Z 310.678,A -85,B 0,C 180,E1 -15353.569,E2 -15353.569} C_VEL
LIN {X 0,Y 319.552,Z 310.681,A -85,B 0,C 180,E1 -15356.694,E2 -15356.694} C_VEL
LIN {X 0,Y 319.553,Z 310.677,A -85,B 0,C 180,E1 -15359.61,E2 -15359.61} C_VEL
LIN {X 0,Y 319.544,Z 310.68,A -85,B 0,C 180,E1 -15362.49,E2 -15362.49} C_VEL
LIN {X 0,Y 319.577,Z 310.677,A -85,B 0,C 180,E1 -15365.299,E2 -15365.299} C_VEL
LIN {X 0,Y 319.572,Z 310.675,A -85,B 0,C 180,E1 -15368.043,E2 -15368.043} C_VEL
LIN {X 0,Y 319.62,Z 310.669,A -85,B 0,C 180,E1 -15372.068,E2 -15372.068} C_VEL
LIN {X 0,Y 319.738,Z 310.654,A -85,B 0,C 180,E1 -15376.005,E2 -15376.005} C_VEL
LIN {X 0,Y 319.74,Z 310.655,A -85,B 0,C 180,E1 -15379.869,E2 -15379.869} C_VEL
LIN {X 0,Y 319.902,Z 310.637,A -85,B 0,C 180,E1 -15383.69,E2 -15383.69} C_VEL
LIN {X 0,Y 319.957,Z 310.632,A -85,B 0,C 180,E1 -15387.478,E2 -15387.478} C_VEL
LIN {X 0,Y 320,Z 310.623,A -85,B 0,C 180,E1 -15391.254,E2 -15391.254} C_VEL
LIN {X 0,Y 319.706,Z 310.663,A -85,B 0,C 180,E1 -15393.777,E2 -15393.777} C_VEL
LIN {X 0,Y 319.874,Z 310.772,A -85,B 0,C 180,E1 -15395.828,E2 -15395.828} C_VEL
LIN {X 0,Y 320.915,Z 316.204,A -85,B 0,C 180,E1 -15397.546,E2 -15397.546} C_VEL
LIN {X 0,Y 328.182,Z 336.91,A -85,B 0,C 180,E1 -15398.582,E2 -15398.582} C_VEL
LIN {X 0,Y 329.815,Z 345.236,A -85,B 0,C 180,E1 -15398.894,E2 -15398.894} C_VEL
LIN {X 0,Y 327.878,Z 424.076,A -85,B 0,C 180,E1 -15400.711,E2 -15400.711} C_VEL
LIN {X 0,Y 327.212,Z 437.963,A -85,B 0,C 180,E1 -15401.298,E2 -15401.298} C_VEL
LIN {X 0,Y 326.419,Z 449.819,A -85,B 0,C 180,E1 -15402.034,E2 -15402.034} C_VEL
LIN {X 0,Y 325.459,Z 461.269,A -85,B 0,C 180,E1 -15402.988,E2 -15402.988} C_VEL
LIN {X 0,Y 324.147,Z 473.259,A -85,B 0,C 180,E1 -15404.273,E2 -15404.273} C_VEL
LIN {X 0,Y 322.965,Z 483.222,A -85,B 0,C 180,E1 -15405.617,E2 -15405.617} C_VEL
LIN {X 0,Y 321.878,Z 492.327,A -85,B 0,C 180,E1 -15407.138,E2 -15407.138} C_VEL
LIN {X 0,Y 320.772,Z 500.661,A -85,B 0,C 180,E1 -15408.849,E2 -15408.849} C_VEL
LIN {X 0,Y 319.928,Z 507.494,A -85,B 0,C 180,E1 -15410.572,E2 -15410.572} C_VEL
LIN {X 0,Y 319.097,Z 514.551,A -85,B 0,C 180,E1 -15412.814,E2 -15412.814} C_VEL
LIN {X 0,Y 318.464,Z 520.103,A -85,B 0,C 180,E1 -15415.202,E2 -15415.202} C_VEL
LIN {X 0,Y 317.902,Z 524.094,A -85,B 0,C 180,E1 -15417.655,E2 -15417.655} C_VEL
LIN {X 0,Y 317.727,Z 525.653,A -85,B 0,C 180,E1 -15419.112,E2 -15419.112} C_VEL
LIN {X 0,Y 317.629,Z 526.723,A -85,B 0,C 180,E1 -15420.584,E2 -15420.584} C_VEL
LIN {X 0,Y 317.622,Z 527.264,A -85,B 0,C 180,E1 -15422.773,E2 -15422.773} C_VEL
LIN {X 0,Y 317.798,Z 526.538,A -85,B 0,C 180,E1 -15425.09,E2 -15425.09} C_VEL
LIN {X 0,Y 318.131,Z 524.59,A -85,B 0,C 180,E1 -15427.316,E2 -15427.316} C_VEL
LIN {X 0,Y 318.743,Z 520.996,A -85,B 0,C 180,E1 -15429.74,E2 -15429.74} C_VEL
LIN {X 0,Y 319.36,Z 517.178,A -85,B 0,C 180,E1 -15431.563,E2 -15431.563} C_VEL
LIN {X 0,Y 320.254,Z 511.617,A -85,B 0,C 180,E1 -15433.598,E2 -15433.598} C_VEL
LIN {X 0,Y 321.474,Z 504.586,A -85,B 0,C 180,E1 -15435.607,E2 -15435.607} C_VEL
LIN {X 0,Y 322.99,Z 495.817,A -85,B 0,C 180,E1 -15437.582,E2 -15437.582} C_VEL
LIN {X 0,Y 324.504,Z 486.302,A -85,B 0,C 180,E1 -15439.279,E2 -15439.279} C_VEL
LIN {X 0,Y 325.88,Z 476.499,A -85,B 0,C 180,E1 -15440.695,E2 -15440.695} C_VEL
LIN {X 0,Y 326.653,Z 471.299,A -85,B 0,C 180,E1 -15441.326,E2 -15441.326} C_VEL
LIN {X 0,Y 326.477,Z 468.071,A -85,B 0,C 180,E1 -15441.74,E2 -15441.74} C_VEL
LIN {X 0,Y 324.441,Z 463.086,A -85,B 0,C 180,E1 -15442.466,E2 -15442.466} C_VEL
LIN {X 0,Y 322.397,Z 457.924,A -85,B 0,C 180,E1 -15443.148,E2 -15443.148} C_VEL
LIN {X 0,Y 322.187,Z 454.426,A -85,B 0,C 180,E1 -15443.482,E2 -15443.482} C_VEL
LIN {X 0,Y 323.271,Z 442.306,A -85,B 0,C 180,E1 -15444.326,E2 -15444.326} C_VEL
LIN {X 0,Y 324.062,Z 429.592,A -85,B 0,C 180,E1 -15444.957,E2 -15444.957} C_VEL
LIN {X 0,Y 324.691,Z 414.745,A -85,B 0,C 180,E1 -15445.384,E2 -15445.384} C_VEL
LIN {X 0,Y 326.593,Z 347.232,A -85,B 0,C 180,E1 -15446.978,E2 -15446.978} C_VEL
LIN {X 0,Y 325.443,Z 342.786,A -85,B 0,C 180,E1 -15447.208,E2 -15447.208} C_VEL
LIN {X 0,Y 319.497,Z 328.679,A -85,B 0,C 180,E1 -15448.189,E2 -15448.189} C_VEL
LIN {X 0,Y 313.877,Z 316.905,A -85,B 0,C 180,E1 -15449.143,E2 -15449.143} C_VEL
LIN {X 0,Y 312.521,Z 311.56,A -85,B 0,C 180,E1 -15450.943,E2 -15450.943} C_VEL
LIN {X 0,Y 312.546,Z 311.559,A -85,B 0,C 180,E1 -15454.707,E2 -15454.707} C_VEL
LIN {X 0,Y 312.496,Z 311.562,A -85,B 0,C 180,E1 -15458.91,E2 -15458.91} C_VEL
LIN {X 0,Y 312.596,Z 311.547,A -85,B 0,C 180,E1 -15461.654,E2 -15461.654} C_VEL
LIN {X 0,Y 312.649,Z 311.54,A -85,B 0,C 180,E1 -15465.684,E2 -15465.684} C_VEL
LIN {X 0,Y 312.641,Z 311.535,A -85,B 0,C 180,E1 -15469.64,E2 -15469.64} C_VEL
LIN {X 0,Y 312.799,Z 311.517,A -85,B 0,C 180,E1 -15472.252,E2 -15472.252} C_VEL
LIN {X 0,Y 312.67,Z 311.536,A -85,B 0,C 180,E1 -15474.842,E2 -15474.842} C_VEL
LIN {X 0,Y 312.945,Z 311.5,A -85,B 0,C 180,E1 -15478.713,E2 -15478.713} C_VEL
LIN {X 0,Y 312.946,Z 311.503,A -85,B 0,C 180,E1 -15481.287,E2 -15481.287} C_VEL
LIN {X 0,Y 312.673,Z 311.536,A -85,B 0,C 180,E1 -15485.158,E2 -15485.158} C_VEL
LIN {X 0,Y 312.816,Z 311.509,A -85,B 0,C 180,E1 -15487.747,E2 -15487.747} C_VEL
LIN {X 0,Y 312.627,Z 311.533,A -85,B 0,C 180,E1 -15491.673,E2 -15491.673} C_VEL
LIN {X 0,Y 312.639,Z 311.54,A -85,B 0,C 180,E1 -15494.876,E2 -15494.876} C_VEL
LIN {X 0,Y 312.595,Z 311.541,A -85,B 0,C 180,E1 -15499.241,E2 -15499.241} C_VEL
LIN {X 0,Y 312.536,Z 311.551,A -85,B 0,C 180,E1 -15502.805,E2 -15502.805} C_VEL
LIN {X 0,Y 312.517,Z 311.553,A -85,B 0,C 180,E1 -15506.729,E2 -15506.729} C_VEL
LIN {X 0,Y 312.508,Z 311.557,A -85,B 0,C 180,E1 -15509.654,E2 -15509.654} C_VEL
LIN {X 0,Y 312.487,Z 311.561,A -85,B 0,C 180,E1 -15513.693,E2 -15513.693} C_VEL
LIN {X 0,Y 312.552,Z 311.553,A -85,B 0,C 180,E1 -15517.382,E2 -15517.382} C_VEL
LIN {X 0,Y 312.507,Z 311.558,A -85,B 0,C 180,E1 -15520.707,E2 -15520.707} C_VEL
LIN {X 0,Y 312.568,Z 311.554,A -85,B 0,C 180,E1 -15524.189,E2 -15524.189} C_VEL
LIN {X 0,Y 312.531,Z 311.559,A -85,B 0,C 180,E1 -15527.909,E2 -15527.909} C_VEL
LIN {X 0,Y 312.536,Z 311.555,A -85,B 0,C 180,E1 -15531.91,E2 -15531.91} C_VEL
LIN {X 0,Y 312.526,Z 311.644,A -85,B 0,C 180,E1 -15535.8,E2 -15535.8} C_VEL
LIN {X 0,Y 315.19,Z 322.167,A -85,B 0,C 180,E1 -15539.154,E2 -15539.154} C_VEL
LIN {X 0,Y 317.197,Z 331.406,A -85,B 0,C 180,E1 -15541.919,E2 -15541.919} C_VEL
LIN {X 0,Y 318.145,Z 336.818,A -85,B 0,C 180,E1 -15543.394,E2 -15543.394} C_VEL
LIN {X 0,Y 321.848,Z 354.245,A -85,B 0,C 180,E1 -15544.245,E2 -15544.245} C_VEL
LIN {X 0,Y 325.083,Z 374.629,A -85,B 0,C 180,E1 -15545.104,E2 -15545.104} C_VEL
LIN {X 0,Y 325.837,Z 380.945,A -85,B 0,C 180,E1 -15545.339,E2 -15545.339} C_VEL
LIN {X 0,Y 323.808,Z 446.779,A -85,B 0,C 180,E1 -15546.91,E2 -15546.91} C_VEL
LIN {X 0,Y 322.832,Z 460.408,A -85,B 0,C 180,E1 -15547.486,E2 -15547.486} C_VEL
LIN {X 0,Y 321.569,Z 473.062,A -85,B 0,C 180,E1 -15548.28,E2 -15548.28} C_VEL
LIN {X 0,Y 320.105,Z 484.733,A -85,B 0,C 180,E1 -15549.272,E2 -15549.272} C_VEL
LIN {X 0,Y 318.467,Z 496.046,A -85,B 0,C 180,E1 -15550.507,E2 -15550.507} C_VEL
LIN {X 0,Y 316.915,Z 506.288,A -85,B 0,C 180,E1 -15551.918,E2 -15551.918} C_VEL
LIN {X 0,Y 315.427,Z 515.679,A -85,B 0,C 180,E1 -15553.534,E2 -15553.534} C_VEL
LIN {X 0,Y 313.977,Z 524.538,A -85,B 0,C 180,E1 -15555.42,E2 -15555.42} C_VEL
LIN {X 0,Y 312.635,Z 531.823,A -85,B 0,C 180,E1 -15557.344,E2 -15557.344} C_VEL
LIN {X 0,Y 311.924,Z 536.765,A -85,B 0,C 180,E1 -15558.964,E2 -15558.964} C_VEL
LIN {X 0,Y 311.3,Z 541.584,A -85,B 0,C 180,E1 -15560.912,E2 -15560.912} C_VEL
LIN {X 0,Y 310.917,Z 545.285,A -85,B 0,C 180,E1 -15562.863,E2 -15562.863} C_VEL
LIN {X 0,Y 310.712,Z 547.97,A -85,B 0,C 180,E1 -15564.814,E2 -15564.814} C_VEL
LIN {X 0,Y 310.718,Z 549.249,A -85,B 0,C 180,E1 -15566.114,E2 -15566.114} C_VEL
LIN {X 0,Y 310.7,Z 550.094,A -85,B 0,C 180,E1 -15567.411,E2 -15567.411} C_VEL
LIN {X 0,Y 310.699,Z 550.518,A -85,B 0,C 180,E1 -15568.708,E2 -15568.708} C_VEL
LIN {X 0,Y 310.759,Z 550.551,A -85,B 0,C 180,E1 -15570.004,E2 -15570.004} C_VEL
LIN {X 0,Y 310.712,Z 550.186,A -85,B 0,C 180,E1 -15571.3,E2 -15571.3} C_VEL
LIN {X 0,Y 310.706,Z 549.396,A -85,B 0,C 180,E1 -15572.597,E2 -15572.597} C_VEL
LIN {X 0,Y 310.741,Z 548.169,A -85,B 0,C 180,E1 -15573.894,E2 -15573.894} C_VEL
LIN {X 0,Y 310.726,Z 545.912,A -85,B 0,C 180,E1 -15575.618,E2 -15575.618} C_VEL
LIN {X 0,Y 311.006,Z 541.864,A -85,B 0,C 180,E1 -15577.796,E2 -15577.796} C_VEL
LIN {X 0,Y 311.388,Z 537.047,A -85,B 0,C 180,E1 -15579.749,E2 -15579.749} C_VEL
LIN {X 0,Y 312.025,Z 530.945,A -85,B 0,C 180,E1 -15581.699,E2 -15581.699} C_VEL
LIN {X 0,Y 313.082,Z 523.349,A -85,B 0,C 180,E1 -15583.636,E2 -15583.636} C_VEL
LIN {X 0,Y 314.122,Z 515.58,A -85,B 0,C 180,E1 -15585.245,E2 -15585.245} C_VEL
LIN {X 0,Y 315.253,Z 506.084,A -85,B 0,C 180,E1 -15586.85,E2 -15586.85} C_VEL
LIN {X 0,Y 316.573,Z 495.547,A -85,B 0,C 180,E1 -15588.278,E2 -15588.278} C_VEL
LIN {X 0,Y 317.941,Z 483.849,A -85,B 0,C 180,E1 -15589.535,E2 -15589.535} C_VEL
LIN {X 0,Y 319.184,Z 471.407,A -85,B 0,C 180,E1 -15590.547,E2 -15590.547} C_VEL
LIN {X 0,Y 320.248,Z 458.384,A -85,B 0,C 180,E1 -15591.316,E2 -15591.316} C_VEL
LIN {X 0,Y 320.984,Z 445.702,A -85,B 0,C 180,E1 -15591.813,E2 -15591.813} C_VEL
LIN {X 0,Y 322.525,Z 379.065,A -85,B 0,C 180,E1 -15593.38,E2 -15593.38} C_VEL
LIN {X 0,Y 317.541,Z 345.25,A -85,B 0,C 180,E1 -15594.574,E2 -15594.574} C_VEL
LIN {X 0,Y 316.43,Z 338.225,A -85,B 0,C 180,E1 -15594.857,E2 -15594.857} C_VEL
LIN {X 0,Y 316.99,Z 333.943,A -85,B 0,C 180,E1 -15595.971,E2 -15595.971} C_VEL
LIN {X 0,Y 315.961,Z 327.288,A -85,B 0,C 180,E1 -15597.849,E2 -15597.849} C_VEL
LIN {X 0,Y 312.98,Z 313.407,A -85,B 0,C 180,E1 -15601.978,E2 -15601.978} C_VEL
LIN {X 0,Y 312.574,Z 311.55,A -85,B 0,C 180,E1 -15602.581,E2 -15602.581} C_VEL
LIN {X 0,Y 312.541,Z 311.555,A -85,B 0,C 180,E1 -15605.951,E2 -15605.951} C_VEL
LIN {X 0,Y 312.51,Z 311.558,A -85,B 0,C 180,E1 -15610.126,E2 -15610.126} C_VEL
LIN {X 0,Y 312.463,Z 311.562,A -85,B 0,C 180,E1 -15613.966,E2 -15613.966} C_VEL
LIN {X 0,Y 312.488,Z 311.559,A -85,B 0,C 180,E1 -15617.92,E2 -15617.92} C_VEL
LIN {X 0,Y 312.502,Z 311.557,A -85,B 0,C 180,E1 -15620.972,E2 -15620.972} C_VEL
LIN {X 0,Y 312.535,Z 311.553,A -85,B 0,C 180,E1 -15624.221,E2 -15624.221} C_VEL
LIN {X 0,Y 312.505,Z 311.556,A -85,B 0,C 180,E1 -15627.334,E2 -15627.334} C_VEL
LIN {X 0,Y 312.572,Z 311.547,A -85,B 0,C 180,E1 -15631.824,E2 -15631.824} C_VEL
LIN {X 0,Y 312.586,Z 311.548,A -85,B 0,C 180,E1 -15634.711,E2 -15634.711} C_VEL
LIN {X 0,Y 312.524,Z 311.558,A -85,B 0,C 180,E1 -15638.912,E2 -15638.912} C_VEL
LIN {X 0,Y 312.577,Z 311.546,A -85,B 0,C 180,E1 -15643.005,E2 -15643.005} C_VEL
LIN {X 0,Y 312.685,Z 311.531,A -85,B 0,C 180,E1 -15645.686,E2 -15645.686} C_VEL
LIN {X 0,Y 312.685,Z 311.534,A -85,B 0,C 180,E1 -15649.641,E2 -15649.641} C_VEL
LIN {X 0,Y 312.844,Z 311.512,A -85,B 0,C 180,E1 -15652.254,E2 -15652.254} C_VEL
LIN {X 0,Y 312.897,Z 311.507,A -85,B 0,C 180,E1 -15653.552,E2 -15653.552} C_VEL
LIN {X 0,Y 312.93,Z 311.499,A -85,B 0,C 180,E1 -15657.426,E2 -15657.426} C_VEL
LIN {X 0,Y 313.049,Z 311.484,A -85,B 0,C 180,E1 -15660,E2 -15660} C_VEL
LIN {X 0,Y 312.929,Z 311.5,A -85,B 0,C 180,E1 -15662.574,E2 -15662.574} C_VEL
LIN {X 0,Y 312.839,Z 311.513,A -85,B 0,C 180,E1 -15666.455,E2 -15666.455} C_VEL
LIN {X 0,Y 312.684,Z 311.531,A -85,B 0,C 180,E1 -15670.359,E2 -15670.359} C_VEL
LIN {X 0,Y 312.668,Z 311.534,A -85,B 0,C 180,E1 -15674.864,E2 -15674.864} C_VEL
LIN {X 0,Y 312.549,Z 311.547,A -85,B 0,C 180,E1 -15679.192,E2 -15679.192} C_VEL
LIN {X 0,Y 312.517,Z 311.553,A -85,B 0,C 180,E1 -15682.775,E2 -15682.775} C_VEL
LIN {X 0,Y 312.479,Z 311.557,A -85,B 0,C 180,E1 -15686.732,E2 -15686.732} C_VEL
LIN {X 0,Y 312.467,Z 311.556,A -85,B 0,C 180,E1 -15689.658,E2 -15689.658} C_VEL
LIN {X 0,Y 312.522,Z 311.548,A -85,B 0,C 180,E1 -15693.688,E2 -15693.688} C_VEL
LIN {X 0,Y 312.512,Z 311.553,A -85,B 0,C 180,E1 -15697.387,E2 -15697.387} C_VEL
LIN {X 0,Y 312.431,Z 311.566,A -85,B 0,C 180,E1 -15700.719,E2 -15700.719} C_VEL
LIN {X 0,Y 312.443,Z 311.564,A -85,B 0,C 180,E1 -15704.211,E2 -15704.211} C_VEL
LIN {X 0,Y 312.431,Z 311.564,A -85,B 0,C 180,E1 -15707.93,E2 -15707.93} C_VEL
LIN {X 0,Y 312.475,Z 311.559,A -85,B 0,C 180,E1 -15711.925,E2 -15711.925} C_VEL
LIN {X 0,Y 312.518,Z 311.554,A -85,B 0,C 180,E1 -15714.216,E2 -15714.216} C_VEL
LIN {X 0,Y 312.487,Z 311.559,A -85,B 0,C 180,E1 -15717.329,E2 -15717.329} C_VEL
LIN {X 0,Y 312.502,Z 311.558,A -85,B 0,C 180,E1 -15721.294,E2 -15721.294} C_VEL
LIN {X 0,Y 312.552,Z 311.553,A -85,B 0,C 180,E1 -15724.705,E2 -15724.705} C_VEL
LIN {X 0,Y 312.53,Z 311.556,A -85,B 0,C 180,E1 -15728.909,E2 -15728.909} C_VEL
LIN {X 0,Y 312.584,Z 311.549,A -85,B 0,C 180,E1 -15733.002,E2 -15733.002} C_VEL
LIN {X 0,Y 312.691,Z 311.534,A -85,B 0,C 180,E1 -15735.683,E2 -15735.683} C_VEL
LIN {X 0,Y 312.69,Z 311.535,A -85,B 0,C 180,E1 -15739.638,E2 -15739.638} C_VEL
LIN {X 0,Y 312.8,Z 311.518,A -85,B 0,C 180,E1 -15742.249,E2 -15742.249} C_VEL
LIN {X 0,Y 312.69,Z 311.533,A -85,B 0,C 180,E1 -15744.838,E2 -15744.838} C_VEL
LIN {X 0,Y 312.981,Z 311.495,A -85,B 0,C 180,E1 -15748.709,E2 -15748.709} C_VEL
LIN {X 0,Y 312.907,Z 311.505,A -85,B 0,C 180,E1 -15752.57,E2 -15752.57} C_VEL
LIN {X 0,Y 312.767,Z 311.7,A -85,B 0,C 180,E1 -15755.475,E2 -15755.475} C_VEL
LIN {X 0,Y 313.813,Z 316.673,A -85,B 0,C 180,E1 -15757.05,E2 -15757.05} C_VEL
LIN {X 0,Y 321.781,Z 339.024,A -85,B 0,C 180,E1 -15758.196,E2 -15758.196} C_VEL
LIN {X 0,Y 323.176,Z 346.358,A -85,B 0,C 180,E1 -15758.475,E2 -15758.475} C_VEL
LIN {X 0,Y 321.168,Z 424.44,A -85,B 0,C 180,E1 -15760.314,E2 -15760.314} C_VEL
LIN {X 0,Y 320.459,Z 438.381,A -85,B 0,C 180,E1 -15760.917,E2 -15760.917} C_VEL
LIN {X 0,Y 319.604,Z 450.99,A -85,B 0,C 180,E1 -15761.731,E2 -15761.731} C_VEL
LIN {X 0,Y 318.527,Z 462.637,A -85,B 0,C 180,E1 -15762.742,E2 -15762.742} C_VEL
LIN {X 0,Y 317.364,Z 473.074,A -85,B 0,C 180,E1 -15763.89,E2 -15763.89} C_VEL
LIN {X 0,Y 316.078,Z 483.411,A -85,B 0,C 180,E1 -15765.305,E2 -15765.305} C_VEL
LIN {X 0,Y 314.96,Z 492.529,A -85,B 0,C 180,E1 -15766.857,E2 -15766.857} C_VEL
LIN {X 0,Y 313.799,Z 500.879,A -85,B 0,C 180,E1 -15768.606,E2 -15768.606} C_VEL
LIN {X 0,Y 312.938,Z 507.714,A -85,B 0,C 180,E1 -15770.365,E2 -15770.365} C_VEL
LIN {X 0,Y 312.075,Z 514.581,A -85,B 0,C 180,E1 -15772.581,E2 -15772.581} C_VEL
LIN {X 0,Y 311.503,Z 519.5,A -85,B 0,C 180,E1 -15774.663,E2 -15774.663} C_VEL
LIN {X 0,Y 310.956,Z 523.329,A -85,B 0,C 180,E1 -15776.867,E2 -15776.867} C_VEL
LIN {X 0,Y 310.718,Z 525.199,A -85,B 0,C 180,E1 -15778.352,E2 -15778.352} C_VEL
LIN {X 0,Y 310.526,Z 527.021,A -85,B 0,C 180,E1 -15780.679,E2 -15780.679} C_VEL
LIN {X 0,Y 310.532,Z 527.504,A -85,B 0,C 180,E1 -15783.134,E2 -15783.134} C_VEL
LIN {X 0,Y 310.751,Z 526.645,A -85,B 0,C 180,E1 -15785.493,E2 -15785.493} C_VEL
LIN {X 0,Y 311.12,Z 524.576,A -85,B 0,C 180,E1 -15787.756,E2 -15787.756} C_VEL
LIN {X 0,Y 311.74,Z 521.293,A -85,B 0,C 180,E1 -15789.958,E2 -15789.958} C_VEL
LIN {X 0,Y 312.63,Z 516.066,A -85,B 0,C 180,E1 -15792.399,E2 -15792.399} C_VEL
LIN {X 0,Y 313.683,Z 510.222,A -85,B 0,C 180,E1 -15794.455,E2 -15794.455} C_VEL
LIN {X 0,Y 314.845,Z 503.936,A -85,B 0,C 180,E1 -15796.212,E2 -15796.212} C_VEL
LIN {X 0,Y 316.251,Z 496.156,A -85,B 0,C 180,E1 -15797.976,E2 -15797.976} C_VEL
LIN {X 0,Y 317.839,Z 486.658,A -85,B 0,C 180,E1 -15799.706,E2 -15799.706} C_VEL
LIN {X 0,Y 319.247,Z 476.983,A -85,B 0,C 180,E1 -15801.135,E2 -15801.135} C_VEL
LIN {X 0,Y 320.737,Z 466.946,A -85,B 0,C 180,E1 -15802.321,E2 -15802.321} C_VEL
LIN {X 0,Y 322.1,Z 455.142,A -85,B 0,C 180,E1 -15803.427,E2 -15803.427} C_VEL
LIN {X 0,Y 322.187,Z 454.426,A -85,B 0,C 180,E1 -15803.482,E2 -15803.482} C_VEL
LIN {X 0,Y 322.246,Z 449.078,A -85,B 0,C 180,E1 -15803.928,E2 -15803.928} C_VEL
LIN {X 0,Y 320.404,Z 440.363,A -85,B 0,C 180,E1 -15804.705,E2 -15804.705} C_VEL
LIN {X 0,Y 318.362,Z 431.441,A -85,B 0,C 180,E1 -15805.382,E2 -15805.382} C_VEL
LIN {X 0,Y 317.977,Z 425.769,A -85,B 0,C 180,E1 -15805.662,E2 -15805.662} C_VEL
LIN {X 0,Y 320.424,Z 348.656,A -85,B 0,C 180,E1 -15807.548,E2 -15807.548} C_VEL
LIN {X 0,Y 319.192,Z 344.606,A -85,B 0,C 180,E1 -15807.783,E2 -15807.783} C_VEL
LIN {X 0,Y 314.002,Z 332.276,A -85,B 0,C 180,E1 -15808.671,E2 -15808.671} C_VEL
LIN {X 0,Y 306.725,Z 317.218,A -85,B 0,C 180,E1 -15809.959,E2 -15809.959} C_VEL
LIN {X 0,Y 305.493,Z 312.435,A -85,B 0,C 180,E1 -15811.58,E2 -15811.58} C_VEL
LIN {X 0,Y 305.533,Z 312.435,A -85,B 0,C 180,E1 -15814.084,E2 -15814.084} C_VEL
LIN {X 0,Y 305.441,Z 312.443,A -85,B 0,C 180,E1 -15818.398,E2 -15818.398} C_VEL
LIN {X 0,Y 305.538,Z 312.426,A -85,B 0,C 180,E1 -15821.214,E2 -15821.214} C_VEL
LIN {X 0,Y 305.595,Z 312.419,A -85,B 0,C 180,E1 -15825.346,E2 -15825.346} C_VEL
LIN {X 0,Y 305.58,Z 312.415,A -85,B 0,C 180,E1 -15829.398,E2 -15829.398} C_VEL
LIN {X 0,Y 305.743,Z 312.397,A -85,B 0,C 180,E1 -15832.072,E2 -15832.072} C_VEL
LIN {X 0,Y 305.641,Z 312.413,A -85,B 0,C 180,E1 -15834.723,E2 -15834.723} C_VEL
LIN {X 0,Y 305.912,Z 312.376,A -85,B 0,C 180,E1 -15838.684,E2 -15838.684} C_VEL
LIN {X 0,Y 305.912,Z 312.379,A -85,B 0,C 180,E1 -15841.316,E2 -15841.316} C_VEL
LIN {X 0,Y 305.644,Z 312.413,A -85,B 0,C 180,E1 -15845.277,E2 -15845.277} C_VEL
LIN {X 0,Y 305.758,Z 312.388,A -85,B 0,C 180,E1 -15847.927,E2 -15847.927} C_VEL
LIN {X 0,Y 305.561,Z 312.412,A -85,B 0,C 180,E1 -15851.947,E2 -15851.947} C_VEL
LIN {X 0,Y 305.579,Z 312.417,A -85,B 0,C 180,E1 -15855.025,E2 -15855.025} C_VEL
LIN {X 0,Y 305.564,Z 312.415,A -85,B 0,C 180,E1 -15859.462,E2 -15859.462} C_VEL
LIN {X 0,Y 305.486,Z 312.429,A -85,B 0,C 180,E1 -15863.059,E2 -15863.059} C_VEL
LIN {X 0,Y 305.511,Z 312.425,A -85,B 0,C 180,E1 -15866.231,E2 -15866.231} C_VEL
LIN {X 0,Y 305.458,Z 312.428,A -85,B 0,C 180,E1 -15869.053,E2 -15869.053} C_VEL
LIN {X 0,Y 305.432,Z 312.441,A -85,B 0,C 180,E1 -15873.521,E2 -15873.521} C_VEL
LIN {X 0,Y 305.491,Z 312.431,A -85,B 0,C 180,E1 -15876.737,E2 -15876.737} C_VEL
LIN {X 0,Y 305.472,Z 312.436,A -85,B 0,C 180,E1 -15880.106,E2 -15880.106} C_VEL
LIN {X 0,Y 305.506,Z 312.432,A -85,B 0,C 180,E1 -15883.641,E2 -15883.641} C_VEL
LIN {X 0,Y 305.497,Z 312.439,A -85,B 0,C 180,E1 -15887.406,E2 -15887.406} C_VEL
LIN {X 0,Y 305.498,Z 312.432,A -85,B 0,C 180,E1 -15891.609,E2 -15891.609} C_VEL
LIN {X 0,Y 305.485,Z 312.516,A -85,B 0,C 180,E1 -15895.107,E2 -15895.107} C_VEL
LIN {X 0,Y 308.293,Z 323.602,A -85,B 0,C 180,E1 -15898.768,E2 -15898.768} C_VEL
LIN {X 0,Y 310.547,Z 334.022,A -85,B 0,C 180,E1 -15901.959,E2 -15901.959} C_VEL
LIN {X 0,Y 310.915,Z 336.152,A -85,B 0,C 180,E1 -15902.585,E2 -15902.585} C_VEL
LIN {X 0,Y 312.747,Z 341.252,A -85,B 0,C 180,E1 -15902.945,E2 -15902.945} C_VEL
LIN {X 0,Y 316.81,Z 362.07,A -85,B 0,C 180,E1 -15903.952,E2 -15903.952} C_VEL
LIN {X 0,Y 319.504,Z 380.713,A -85,B 0,C 180,E1 -15904.73,E2 -15904.73} C_VEL
LIN {X 0,Y 317.558,Z 444.666,A -85,B 0,C 180,E1 -15906.284,E2 -15906.284} C_VEL
LIN {X 0,Y 316.672,Z 457.646,A -85,B 0,C 180,E1 -15906.807,E2 -15906.807} C_VEL
LIN {X 0,Y 315.412,Z 470.437,A -85,B 0,C 180,E1 -15907.575,E2 -15907.575} C_VEL
LIN {X 0,Y 313.947,Z 481.897,A -85,B 0,C 180,E1 -15908.502,E2 -15908.502} C_VEL
LIN {X 0,Y 312.249,Z 493.714,A -85,B 0,C 180,E1 -15909.76,E2 -15909.76} C_VEL
